// TIA Portal V16 export
// export: Created 2021-11-12T13:31:00.4796607Z, ExportSetting WithDefaults, DisplayName Totally Integrated Automation Portal, DisplayVersion V16 Update 3, DisplayName TIA Portal Version Control Interface, DisplayVersion V16 Update 2, DisplayName TIA Portal Openness, DisplayVersion V16 Update 3, DisplayName SINAMICS Startdrive Advanced, DisplayVersion V16 Update 5, DisplayName SINAMICS Startdrive G130, G150, S120, S150, SINAMICS MV, S210, DisplayVersion V16 Update 5, DisplayName SINAMICS Startdrive G110M, G120, G120C, G120D, G120P, G115D, DisplayVersion V16 Update 5, DisplayName STEP 7 Professional, DisplayVersion V16 Update 3, DisplayName STEP 7 Safety, DisplayVersion V16, DisplayName WinCC UA Professional, DisplayVersion V16 Update 3
FUNCTION_BLOCK "Safety_Aux"   // FB66, LAD
{ S7_Optimized_Access := 'TRUE' }
VERSION : 0.1
// stored: AutoNumber true, IsIECCheckEnabled false, IsRetainMemResEnabled false, MemoryReserve 100, SetENOAutomatically false, UDAEnableTagReadback false
   VAR
      "SF_100+RU01-QQ01" : "STD_EuchnerDoor";
      "SF_100+RU01-QQ02" { S7_SetPoint := 'True'} : "STD_EuchnerDoor";
      "SF_100+RU01-QQ03" { S7_SetPoint := 'True'} : "STD_EuchnerDoor";
      "SF_100+RU01-QQ04" { S7_SetPoint := 'True'} : "STD_EuchnerDoor";
      "SF_100+RU01-QQ05" { S7_SetPoint := 'True'} : "STD_EuchnerDoor";
      "SF_100+RU01-QQ06" { S7_SetPoint := 'True'} : "STD_EuchnerDoor";
      "SF_100+RU01-QQ07" { S7_SetPoint := 'True'} : "STD_EuchnerDoor";
      "SF_100+RU01-QQ08" { S7_SetPoint := 'True'} : "STD_EuchnerDoor";
      "SF_200+RU01-QQ01" { S7_SetPoint := 'True'} : "STD_EuchnerDoor";
      "SF_200+RU01-QQ02" { S7_SetPoint := 'True'} : "STD_EuchnerDoor";
      "SF_200+RU01-QQ03" { S7_SetPoint := 'True'} : "STD_EuchnerDoor";
      "SF_200+RU01-QQ04" { S7_SetPoint := 'True'} : "STD_EuchnerDoor";
      "SF_200+RU01-QQ05" { S7_SetPoint := 'True'} : "STD_EuchnerDoor";
      "SF_100+RU01-KF01" { S7_SetPoint := 'True'} : "STD_EuchnerSafetySwitch2MBM";
      "SF_100+RU01-KF02" { S7_SetPoint := 'True'} : "STD_EuchnerSafetySwitch2MBM";
      "SF_100+RU01-KF03" { S7_SetPoint := 'True'} : "STD_EuchnerSafetySwitch2MBM";
      "SF_200+RU01-KF01" { S7_SetPoint := 'True'} : "STD_EuchnerSafetySwitch2MBM";
      "SF_200+RU01-KF02" { S7_SetPoint := 'True'} : "STD_EuchnerSafetySwitch2MBM";
      "SF_200+RU01-KF03" { S7_SetPoint := 'True'} : "STD_EuchnerSafetySwitch2MBM";
      "SF_200+RU01-KF04" { S7_SetPoint := 'True'} : "STD_EuchnerSafetySwitch2MBM";
      SF_KAS1_ES { S7_SetPoint := 'True'} : "STD_DI_Mon";
      SF_KAS2_ES { S7_SetPoint := 'True'} : "STD_DI_Mon";
      SF_BSN1_2_ES { S7_SetPoint := 'True'} : "STD_DI_Mon";
      SF_BSN3_ES { S7_SetPoint := 'True'} : "STD_DI_Mon";
      SF_BSN4_5_ES { S7_SetPoint := 'True'} : "STD_DI_Mon";
      SF_SCH1_ES { S7_SetPoint := 'True'} : "STD_DI_Mon";
      SF_THM1_ES { S7_SetPoint := 'True'} : "STD_DI_Mon";
      SF_THM2_ES { S7_SetPoint := 'True'} : "STD_DI_Mon";
      "SF_000UH10-SF01_ES" { S7_SetPoint := 'True'} : "STD_DI_Mon";
      "SF_000UH11-SF01_ES" { S7_SetPoint := 'True'} : "STD_DI_Mon";
      "SF_100UH11-SF01_ES" { S7_SetPoint := 'True'} : "STD_DI_Mon";
      "SF_100UH12-SF01_ES" { S7_SetPoint := 'True'} : "STD_DI_Mon";
      "SF_100UH13-SF01_ES" { S7_SetPoint := 'True'} : "STD_DI_Mon";
      "SF_100UF01-SF01_ES" { S7_SetPoint := 'True'} : "STD_DI_Mon";
      "SF_200UH11-SF01_ES" { S7_SetPoint := 'True'} : "STD_DI_Mon";
      "SF_210UF01-SF01_ES" { S7_SetPoint := 'True'} : "STD_DI_Mon";
      "SF_220UF01-SF01_ES" { S7_SetPoint := 'True'} : "STD_DI_Mon";
      "SF_230UF01-SF01_ES" { S7_SetPoint := 'True'} : "STD_DI_Mon";
      "SF_200UF01-SF01_ES" { S7_SetPoint := 'True'} : "STD_DI_Mon";
      "SF_300UH11-SF01_ES" { S7_SetPoint := 'True'} : "STD_DI_Mon";
      "SF_310UH31-SF01_ES" { S7_SetPoint := 'True'} : "STD_DI_Mon";
      "SF_330UF01-SF01_ES" { S7_SetPoint := 'True'} : "STD_DI_Mon";
      "SF_400UH11-SF01_ES" { S7_SetPoint := 'True'} : "STD_DI_Mon";
      "SF_410UH31-SF01_ES" { S7_SetPoint := 'True'} : "STD_DI_Mon";
      "SF_420UH31-SF01_ES" { S7_SetPoint := 'True'} : "STD_DI_Mon";
      "SF_430UF01-SF01_ES" { S7_SetPoint := 'True'} : "STD_DI_Mon";
      SF_100QQ01_ES { S7_SetPoint := 'True'} : "STD_DI_Mon";
      SF_100QQ02_ES { S7_SetPoint := 'True'} : "STD_DI_Mon";
      SF_100QQ03_ES { S7_SetPoint := 'True'} : "STD_DI_Mon";
      SF_100QQ04_ES { S7_SetPoint := 'True'} : "STD_DI_Mon";
      SF_100QQ05_ES { S7_SetPoint := 'True'} : "STD_DI_Mon";
      SF_100QQ06_ES { S7_SetPoint := 'True'} : "STD_DI_Mon";
      SF_100QQ07_ES { S7_SetPoint := 'True'} : "STD_DI_Mon";
      SF_100QQ08_ES { S7_SetPoint := 'True'} : "STD_DI_Mon";
      SF_200QQ01_ES { S7_SetPoint := 'True'} : "STD_DI_Mon";
      SF_200QQ02_ES { S7_SetPoint := 'True'} : "STD_DI_Mon";
      SF_200QQ03_ES { S7_SetPoint := 'True'} : "STD_DI_Mon";
      SF_200QQ04_ES { S7_SetPoint := 'True'} : "STD_DI_Mon";
      SF_200QQ05_ES { S7_SetPoint := 'True'} : "STD_DI_Mon";
      SF_1R1RC01_ES { S7_SetPoint := 'True'} : "STD_DI_Mon";
      SF_1R2RC01_ES { S7_SetPoint := 'True'} : "STD_DI_Mon";
      SF_1R3RC01_ES { S7_SetPoint := 'True'} : "STD_DI_Mon";
      SF_1R4RC01_ES { S7_SetPoint := 'True'} : "STD_DI_Mon";
      SF_1R5RC01_ES { S7_SetPoint := 'True'} : "STD_DI_Mon";
      SF_1R6RC01_ES { S7_SetPoint := 'True'} : "STD_DI_Mon";
      SF_2R1RC01_ES { S7_SetPoint := 'True'} : "STD_DI_Mon";
      SF_2R2RC01_ES { S7_SetPoint := 'True'} : "STD_DI_Mon";
      "SF_000UH01-KF31" { S7_SetPoint := 'True'} : "STD_DI_Mon";
      "SF_000UH01-KF32" { S7_SetPoint := 'True'} : "STD_DI_Mon";
      "SF_000UH01-KF33" { S7_SetPoint := 'True'} : "STD_DI_Mon";
      "SF_000UH01-KF41" { S7_SetPoint := 'True'} : "STD_DI_Mon";
      "SF_000UH11-KF31" { S7_SetPoint := 'True'} : "STD_DI_Mon";
      "SF_000UH11-KF32" { S7_SetPoint := 'True'} : "STD_DI_Mon";
      "SF_100UH11-KF31" { S7_SetPoint := 'True'} : "STD_DI_Mon";
      "SF_100UH12-KF31" { S7_SetPoint := 'True'} : "STD_DI_Mon";
      "SF_100UH13-KF31" { S7_SetPoint := 'True'} : "STD_DI_Mon";
      "SF_100UH13-KF32" { S7_SetPoint := 'True'} : "STD_DI_Mon";
      "SF_200UH11-KF31" { S7_SetPoint := 'True'} : "STD_DI_Mon";
      "SF_300UH11-KF31" { S7_SetPoint := 'True'} : "STD_DI_Mon";
      "SF_310UH31-KF31" { S7_SetPoint := 'True'} : "STD_DI_Mon";
      "SF_400UH11-KF31" { S7_SetPoint := 'True'} : "STD_DI_Mon";
      "SF_410UH31-KF31" { S7_SetPoint := 'True'} : "STD_DI_Mon";
      "SF_420UH31-KF31" { S7_SetPoint := 'True'} : "STD_DI_Mon";
      "SF_100RU01-KF01" { S7_SetPoint := 'True'} : "STD_DI_Mon";
      "SF_100RU01-KF02" { S7_SetPoint := 'True'} : "STD_DI_Mon";
      "SF_100RU01-KF03" { S7_SetPoint := 'True'} : "STD_DI_Mon";
      "SF_200RU01-KF01" { S7_SetPoint := 'True'} : "STD_DI_Mon";
      "SF_200RU01-KF02" { S7_SetPoint := 'True'} : "STD_DI_Mon";
      "SF_200RU01-KF03" { S7_SetPoint := 'True'} : "STD_DI_Mon";
      "SF_200RU01-KF04" { S7_SetPoint := 'True'} : "STD_DI_Mon";
   END_VAR
   VAR_TEMP
      TS_AckSafety : "UDT_AckSafety1";   // Acknowledgement groups
      TB1UlckEn100 : Bool;
      TB1UlckEn101 : Bool;
      TB1UlckEn102 : Bool;
      TB1UlckEn103 : Bool;
      TB1UlckEn104 : Bool;
      TB1UlckEn105 : Bool;
      TB1UlckEn200 : Bool;
      TB1Fit1 : Bool;
   END_VAR
   VAR_TEMP   // added for the SCL form of the ladder/FBD networks
      _w1 : Bool;
      _w2 : Bool;
      _w3 : Bool;
      _w4 : Bool;
      _w5 : Bool;
      _w6 : Bool;
      _w7 : Bool;
      _w8 : Bool;
   END_VAR
BEGIN

REGION Network 1: *************** Resets ***************
END_REGION

REGION Network 2: Safety acknowledge Group01
   // Group01 - zone 100 buttons included panel 000-UH11, panel 000-UH10
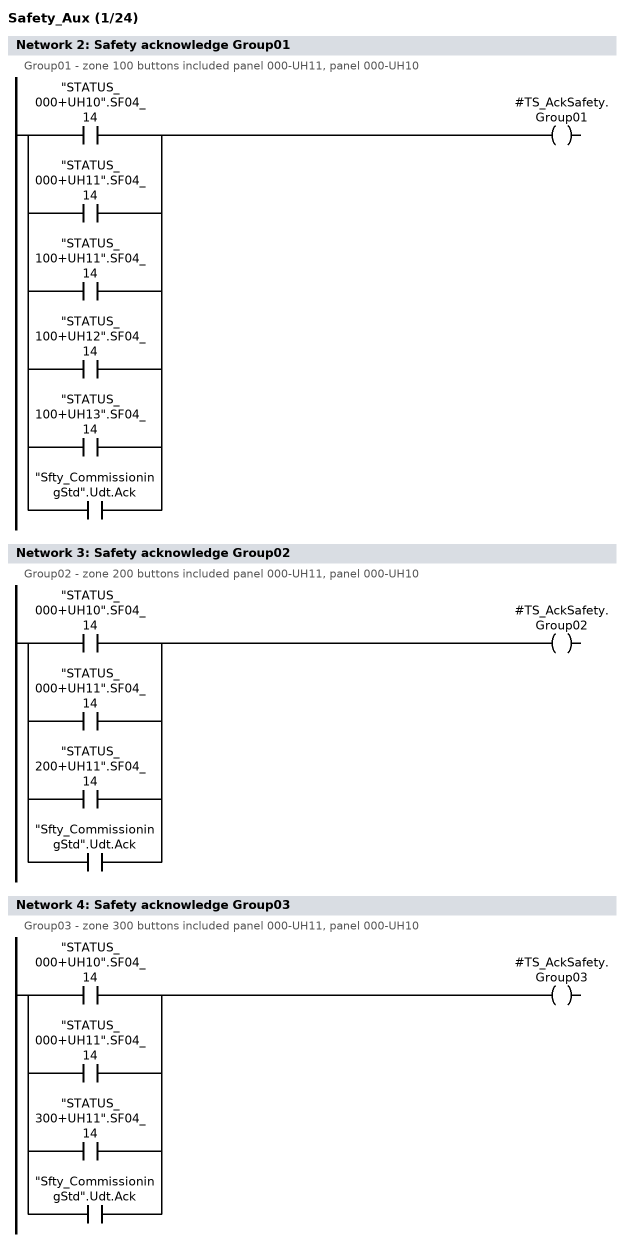
   RUNG wire#powerrail
      Contact( "STATUS_000+UH10".SF04_14 )
      wire#w1
      Coil( #TS_AckSafety.Group01 )
   END_RUNG
   RUNG wire#powerrail
      Contact( "STATUS_000+UH11".SF04_14 )
   END_RUNG wire#w1
   RUNG wire#powerrail
      Contact( "STATUS_100+UH11".SF04_14 )
   END_RUNG wire#w1
   RUNG wire#powerrail
      Contact( "STATUS_100+UH12".SF04_14 )
   END_RUNG wire#w1
   RUNG wire#powerrail
      Contact( "STATUS_100+UH13".SF04_14 )
   END_RUNG wire#w1
   RUNG wire#powerrail
      Contact( "Sfty_CommissioningStd".Udt.Ack )
   END_RUNG wire#w1
   // the same network as SCL:
   #TS_AckSafety.Group01 := "STATUS_000+UH10".SF04_14 OR "STATUS_000+UH11".SF04_14 OR "STATUS_100+UH11".SF04_14 OR "STATUS_100+UH12".SF04_14 OR "STATUS_100+UH13".SF04_14 OR "Sfty_CommissioningStd".Udt.Ack;
END_REGION

REGION Network 3: Safety acknowledge Group02
   // Group02 - zone 200 buttons included panel 000-UH11, panel 000-UH10
   RUNG wire#powerrail
      Contact( "STATUS_000+UH10".SF04_14 )
      wire#w1
      Coil( #TS_AckSafety.Group02 )
   END_RUNG
   RUNG wire#powerrail
      Contact( "STATUS_000+UH11".SF04_14 )
   END_RUNG wire#w1
   RUNG wire#powerrail
      Contact( "STATUS_200+UH11".SF04_14 )
   END_RUNG wire#w1
   RUNG wire#powerrail
      Contact( "Sfty_CommissioningStd".Udt.Ack )
   END_RUNG wire#w1
   // the same network as SCL:
   #TS_AckSafety.Group02 := "STATUS_000+UH10".SF04_14 OR "STATUS_000+UH11".SF04_14 OR "STATUS_200+UH11".SF04_14 OR "Sfty_CommissioningStd".Udt.Ack;
END_REGION

REGION Network 4: Safety acknowledge Group03
   // Group03 - zone 300 buttons included panel 000-UH11, panel 000-UH10
   RUNG wire#powerrail
      Contact( "STATUS_000+UH10".SF04_14 )
      wire#w1
      Coil( #TS_AckSafety.Group03 )
   END_RUNG
   RUNG wire#powerrail
      Contact( "STATUS_000+UH11".SF04_14 )
   END_RUNG wire#w1
   RUNG wire#powerrail
      Contact( "STATUS_300+UH11".SF04_14 )
   END_RUNG wire#w1
   RUNG wire#powerrail
      Contact( "Sfty_CommissioningStd".Udt.Ack )
   END_RUNG wire#w1
   // the same network as SCL:
   #TS_AckSafety.Group03 := "STATUS_000+UH10".SF04_14 OR "STATUS_000+UH11".SF04_14 OR "STATUS_300+UH11".SF04_14 OR "Sfty_CommissioningStd".Udt.Ack;
END_REGION

REGION Network 5: Safety acknowledge Group04
   // Group04 - zone 400 buttons included panel 000-UH11, panel 000-UH10
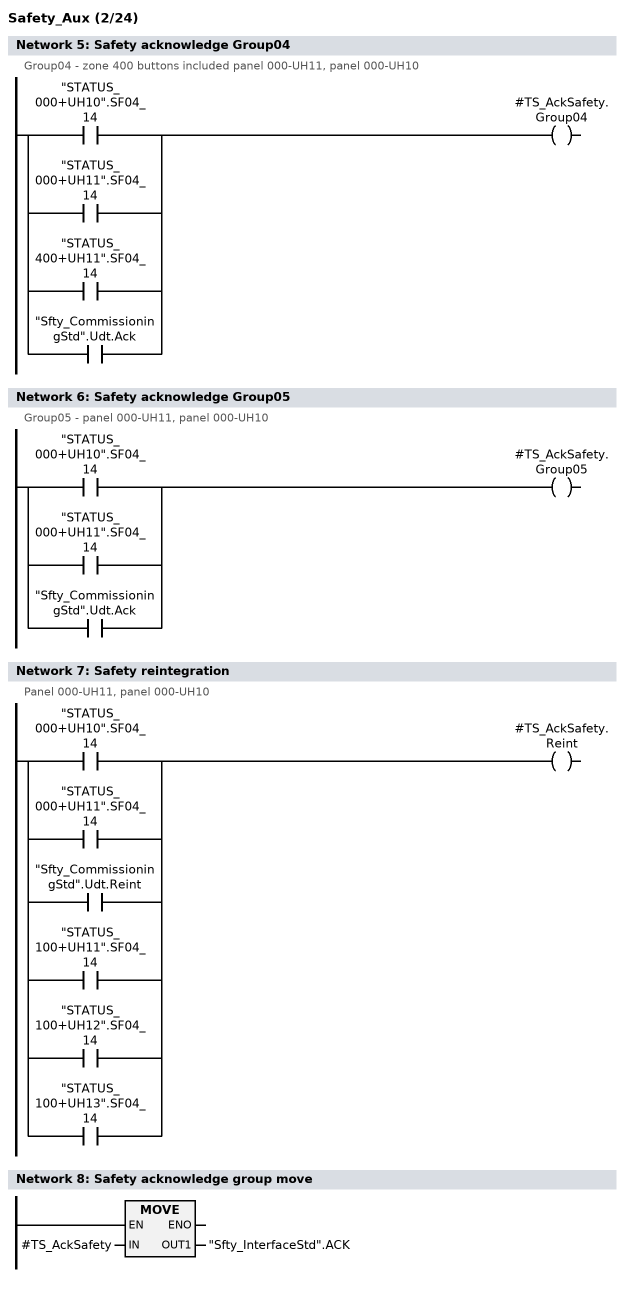
   RUNG wire#powerrail
      Contact( "STATUS_000+UH10".SF04_14 )
      wire#w1
      Coil( #TS_AckSafety.Group04 )
   END_RUNG
   RUNG wire#powerrail
      Contact( "STATUS_000+UH11".SF04_14 )
   END_RUNG wire#w1
   RUNG wire#powerrail
      Contact( "STATUS_400+UH11".SF04_14 )
   END_RUNG wire#w1
   RUNG wire#powerrail
      Contact( "Sfty_CommissioningStd".Udt.Ack )
   END_RUNG wire#w1
   // the same network as SCL:
   #TS_AckSafety.Group04 := "STATUS_000+UH10".SF04_14 OR "STATUS_000+UH11".SF04_14 OR "STATUS_400+UH11".SF04_14 OR "Sfty_CommissioningStd".Udt.Ack;
END_REGION

REGION Network 6: Safety acknowledge Group05
   // Group05 - panel 000-UH11, panel 000-UH10
   RUNG wire#powerrail
      Contact( "STATUS_000+UH10".SF04_14 )
      wire#w1
      Coil( #TS_AckSafety.Group05 )
   END_RUNG
   RUNG wire#powerrail
      Contact( "STATUS_000+UH11".SF04_14 )
   END_RUNG wire#w1
   RUNG wire#powerrail
      Contact( "Sfty_CommissioningStd".Udt.Ack )
   END_RUNG wire#w1
   // the same network as SCL:
   #TS_AckSafety.Group05 := "STATUS_000+UH10".SF04_14 OR "STATUS_000+UH11".SF04_14 OR "Sfty_CommissioningStd".Udt.Ack;
END_REGION

REGION Network 7: Safety reintegration
   // Panel 000-UH11, panel 000-UH10
   RUNG wire#powerrail
      Contact( "STATUS_000+UH10".SF04_14 )
      wire#w1
      Coil( #TS_AckSafety.Reint )
   END_RUNG
   RUNG wire#powerrail
      Contact( "STATUS_000+UH11".SF04_14 )
   END_RUNG wire#w1
   RUNG wire#powerrail
      Contact( "Sfty_CommissioningStd".Udt.Reint )
   END_RUNG wire#w1
   RUNG wire#powerrail
      Contact( "STATUS_100+UH11".SF04_14 )
   END_RUNG wire#w1
   RUNG wire#powerrail
      Contact( "STATUS_100+UH12".SF04_14 )
   END_RUNG wire#w1
   RUNG wire#powerrail
      Contact( "STATUS_100+UH13".SF04_14 )
   END_RUNG wire#w1
   // the same network as SCL:
   #TS_AckSafety.Reint := "STATUS_000+UH10".SF04_14 OR "STATUS_000+UH11".SF04_14 OR "Sfty_CommissioningStd".Udt.Reint OR "STATUS_100+UH11".SF04_14 OR "STATUS_100+UH12".SF04_14 OR "STATUS_100+UH13".SF04_14;
END_REGION

REGION Network 8: Safety acknowledge group move
   RUNG wire#powerrail
      Move(in := #TS_AckSafety, out1 => "Sfty_InterfaceStd".ACK)
   END_RUNG
   // the same network as SCL:
   "Sfty_InterfaceStd".ACK := #TS_AckSafety;
END_REGION

REGION Network 9: *************** Enable unlock gates ***************
END_REGION

REGION Network 10: Zone 100 - enable unlock gates
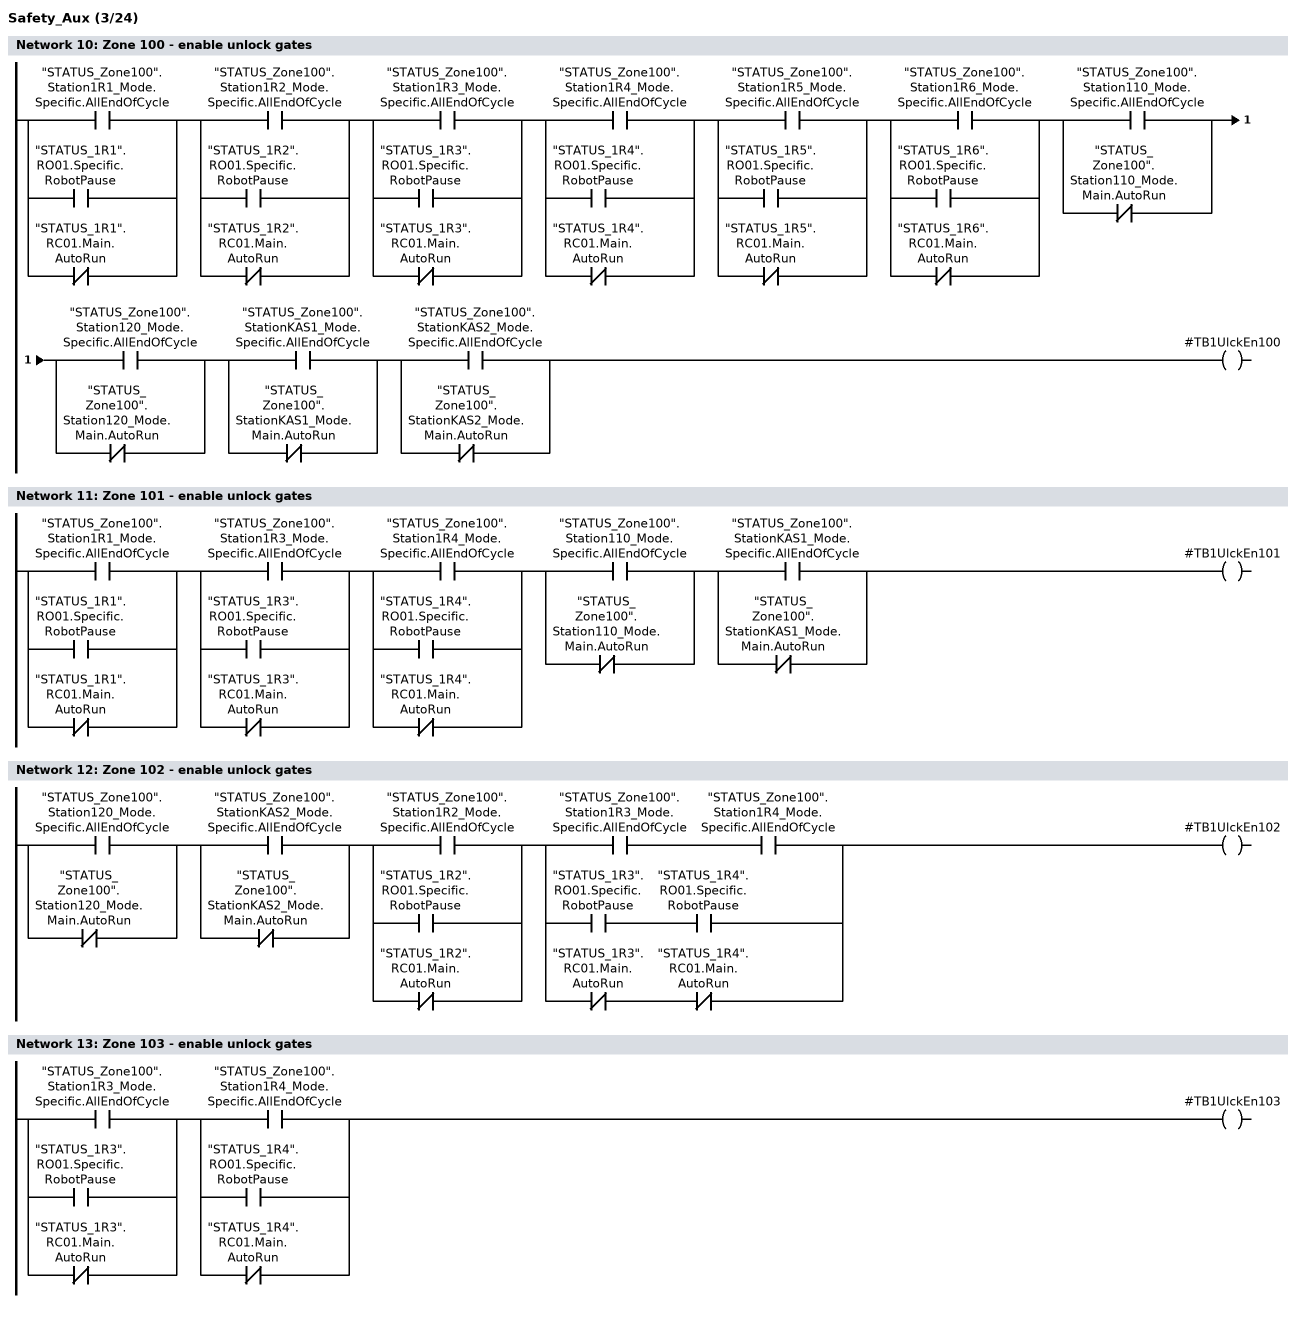
   RUNG wire#powerrail
      Contact( "STATUS_Zone100".Station1R1_Mode.Specific.AllEndOfCycle )
      wire#w1
      Contact( "STATUS_Zone100".Station1R2_Mode.Specific.AllEndOfCycle )
      wire#w2
      Contact( "STATUS_Zone100".Station1R3_Mode.Specific.AllEndOfCycle )
      wire#w3
      Contact( "STATUS_Zone100".Station1R4_Mode.Specific.AllEndOfCycle )
      wire#w4
      Contact( "STATUS_Zone100".Station1R5_Mode.Specific.AllEndOfCycle )
      wire#w5
      Contact( "STATUS_Zone100".Station1R6_Mode.Specific.AllEndOfCycle )
      wire#w6
      Contact( "STATUS_Zone100".Station110_Mode.Specific.AllEndOfCycle )
      wire#w7
      Contact( "STATUS_Zone100".Station120_Mode.Specific.AllEndOfCycle )
      wire#w8
      Contact( "STATUS_Zone100".StationKAS1_Mode.Specific.AllEndOfCycle )
      wire#w9
      Contact( "STATUS_Zone100".StationKAS2_Mode.Specific.AllEndOfCycle )
      wire#w10
      Coil( #TB1UlckEn100 )
   END_RUNG
   RUNG wire#powerrail
      Contact( "STATUS_1R1".RO01.Specific.RobotPause )
   END_RUNG wire#w1
   RUNG wire#powerrail
      I_Contact( "STATUS_1R1".RC01.Main.AutoRun )
   END_RUNG wire#w1
   RUNG wire#w1
      Contact( "STATUS_1R2".RO01.Specific.RobotPause )
   END_RUNG wire#w2
   RUNG wire#w1
      I_Contact( "STATUS_1R2".RC01.Main.AutoRun )
   END_RUNG wire#w2
   RUNG wire#w2
      Contact( "STATUS_1R3".RO01.Specific.RobotPause )
   END_RUNG wire#w3
   RUNG wire#w2
      I_Contact( "STATUS_1R3".RC01.Main.AutoRun )
   END_RUNG wire#w3
   RUNG wire#w3
      Contact( "STATUS_1R4".RO01.Specific.RobotPause )
   END_RUNG wire#w4
   RUNG wire#w3
      I_Contact( "STATUS_1R4".RC01.Main.AutoRun )
   END_RUNG wire#w4
   RUNG wire#w4
      Contact( "STATUS_1R5".RO01.Specific.RobotPause )
   END_RUNG wire#w5
   RUNG wire#w4
      I_Contact( "STATUS_1R5".RC01.Main.AutoRun )
   END_RUNG wire#w5
   RUNG wire#w5
      Contact( "STATUS_1R6".RO01.Specific.RobotPause )
   END_RUNG wire#w6
   RUNG wire#w5
      I_Contact( "STATUS_1R6".RC01.Main.AutoRun )
   END_RUNG wire#w6
   RUNG wire#w6
      I_Contact( "STATUS_Zone100".Station110_Mode.Main.AutoRun )
   END_RUNG wire#w7
   RUNG wire#w7
      I_Contact( "STATUS_Zone100".Station120_Mode.Main.AutoRun )
   END_RUNG wire#w8
   RUNG wire#w8
      I_Contact( "STATUS_Zone100".StationKAS1_Mode.Main.AutoRun )
   END_RUNG wire#w9
   RUNG wire#w9
      I_Contact( "STATUS_Zone100".StationKAS2_Mode.Main.AutoRun )
   END_RUNG wire#w10
   // the same network as SCL:
   #TB1UlckEn100 := ("STATUS_Zone100".Station1R1_Mode.Specific.AllEndOfCycle OR "STATUS_1R1".RO01.Specific.RobotPause OR NOT "STATUS_1R1".RC01.Main.AutoRun) AND ("STATUS_Zone100".Station1R2_Mode.Specific.AllEndOfCycle OR "STATUS_1R2".RO01.Specific.RobotPause OR NOT "STATUS_1R2".RC01.Main.AutoRun) AND ("STATUS_Zone100".Station1R3_Mode.Specific.AllEndOfCycle OR "STATUS_1R3".RO01.Specific.RobotPause OR NOT "STATUS_1R3".RC01.Main.AutoRun) AND ("STATUS_Zone100".Station1R4_Mode.Specific.AllEndOfCycle OR "STATUS_1R4".RO01.Specific.RobotPause OR NOT "STATUS_1R4".RC01.Main.AutoRun) AND ("STATUS_Zone100".Station1R5_Mode.Specific.AllEndOfCycle OR "STATUS_1R5".RO01.Specific.RobotPause OR NOT "STATUS_1R5".RC01.Main.AutoRun) AND ("STATUS_Zone100".Station1R6_Mode.Specific.AllEndOfCycle OR "STATUS_1R6".RO01.Specific.RobotPause OR NOT "STATUS_1R6".RC01.Main.AutoRun) AND ("STATUS_Zone100".Station110_Mode.Specific.AllEndOfCycle OR NOT "STATUS_Zone100".Station110_Mode.Main.AutoRun) AND ("STATUS_Zone100".Station120_Mode.Specific.AllEndOfCycle OR NOT "STATUS_Zone100".Station120_Mode.Main.AutoRun) AND ("STATUS_Zone100".StationKAS1_Mode.Specific.AllEndOfCycle OR NOT "STATUS_Zone100".StationKAS1_Mode.Main.AutoRun) AND ("STATUS_Zone100".StationKAS2_Mode.Specific.AllEndOfCycle OR NOT "STATUS_Zone100".StationKAS2_Mode.Main.AutoRun);
END_REGION

REGION Network 11: Zone 101 - enable unlock gates
   RUNG wire#powerrail
      Contact( "STATUS_Zone100".Station1R1_Mode.Specific.AllEndOfCycle )
      wire#w1
      Contact( "STATUS_Zone100".Station1R3_Mode.Specific.AllEndOfCycle )
      wire#w2
      Contact( "STATUS_Zone100".Station1R4_Mode.Specific.AllEndOfCycle )
      wire#w3
      Contact( "STATUS_Zone100".Station110_Mode.Specific.AllEndOfCycle )
      wire#w4
      Contact( "STATUS_Zone100".StationKAS1_Mode.Specific.AllEndOfCycle )
      wire#w5
      Coil( #TB1UlckEn101 )
   END_RUNG
   RUNG wire#powerrail
      Contact( "STATUS_1R1".RO01.Specific.RobotPause )
   END_RUNG wire#w1
   RUNG wire#powerrail
      I_Contact( "STATUS_1R1".RC01.Main.AutoRun )
   END_RUNG wire#w1
   RUNG wire#w1
      Contact( "STATUS_1R3".RO01.Specific.RobotPause )
   END_RUNG wire#w2
   RUNG wire#w1
      I_Contact( "STATUS_1R3".RC01.Main.AutoRun )
   END_RUNG wire#w2
   RUNG wire#w2
      Contact( "STATUS_1R4".RO01.Specific.RobotPause )
   END_RUNG wire#w3
   RUNG wire#w2
      I_Contact( "STATUS_1R4".RC01.Main.AutoRun )
   END_RUNG wire#w3
   RUNG wire#w3
      I_Contact( "STATUS_Zone100".Station110_Mode.Main.AutoRun )
   END_RUNG wire#w4
   RUNG wire#w4
      I_Contact( "STATUS_Zone100".StationKAS1_Mode.Main.AutoRun )
   END_RUNG wire#w5
   // the same network as SCL:
   #TB1UlckEn101 := ("STATUS_Zone100".Station1R1_Mode.Specific.AllEndOfCycle OR "STATUS_1R1".RO01.Specific.RobotPause OR NOT "STATUS_1R1".RC01.Main.AutoRun) AND ("STATUS_Zone100".Station1R3_Mode.Specific.AllEndOfCycle OR "STATUS_1R3".RO01.Specific.RobotPause OR NOT "STATUS_1R3".RC01.Main.AutoRun) AND ("STATUS_Zone100".Station1R4_Mode.Specific.AllEndOfCycle OR "STATUS_1R4".RO01.Specific.RobotPause OR NOT "STATUS_1R4".RC01.Main.AutoRun) AND ("STATUS_Zone100".Station110_Mode.Specific.AllEndOfCycle OR NOT "STATUS_Zone100".Station110_Mode.Main.AutoRun) AND ("STATUS_Zone100".StationKAS1_Mode.Specific.AllEndOfCycle OR NOT "STATUS_Zone100".StationKAS1_Mode.Main.AutoRun);
END_REGION

REGION Network 12: Zone 102 - enable unlock gates
   RUNG wire#powerrail
      Contact( "STATUS_Zone100".Station120_Mode.Specific.AllEndOfCycle )
      wire#w1
      Contact( "STATUS_Zone100".StationKAS2_Mode.Specific.AllEndOfCycle )
      wire#w2
      Contact( "STATUS_Zone100".Station1R2_Mode.Specific.AllEndOfCycle )
      wire#w3
      Contact( "STATUS_Zone100".Station1R3_Mode.Specific.AllEndOfCycle )
      Contact( "STATUS_Zone100".Station1R4_Mode.Specific.AllEndOfCycle )
      wire#w4
      Coil( #TB1UlckEn102 )
   END_RUNG
   RUNG wire#powerrail
      I_Contact( "STATUS_Zone100".Station120_Mode.Main.AutoRun )
   END_RUNG wire#w1
   RUNG wire#w1
      I_Contact( "STATUS_Zone100".StationKAS2_Mode.Main.AutoRun )
   END_RUNG wire#w2
   RUNG wire#w2
      Contact( "STATUS_1R2".RO01.Specific.RobotPause )
   END_RUNG wire#w3
   RUNG wire#w2
      I_Contact( "STATUS_1R2".RC01.Main.AutoRun )
   END_RUNG wire#w3
   RUNG wire#w3
      Contact( "STATUS_1R3".RO01.Specific.RobotPause )
      Contact( "STATUS_1R4".RO01.Specific.RobotPause )
   END_RUNG wire#w4
   RUNG wire#w3
      I_Contact( "STATUS_1R3".RC01.Main.AutoRun )
      I_Contact( "STATUS_1R4".RC01.Main.AutoRun )
   END_RUNG wire#w4
   // the same network as SCL:
   #TB1UlckEn102 := ("STATUS_Zone100".Station120_Mode.Specific.AllEndOfCycle OR NOT "STATUS_Zone100".Station120_Mode.Main.AutoRun) AND ("STATUS_Zone100".StationKAS2_Mode.Specific.AllEndOfCycle OR NOT "STATUS_Zone100".StationKAS2_Mode.Main.AutoRun) AND ("STATUS_Zone100".Station1R2_Mode.Specific.AllEndOfCycle OR "STATUS_1R2".RO01.Specific.RobotPause OR NOT "STATUS_1R2".RC01.Main.AutoRun) AND (("STATUS_Zone100".Station1R3_Mode.Specific.AllEndOfCycle AND "STATUS_Zone100".Station1R4_Mode.Specific.AllEndOfCycle) OR ("STATUS_1R3".RO01.Specific.RobotPause AND "STATUS_1R4".RO01.Specific.RobotPause) OR (NOT "STATUS_1R3".RC01.Main.AutoRun AND NOT "STATUS_1R4".RC01.Main.AutoRun));
END_REGION

REGION Network 13: Zone 103 - enable unlock gates
   RUNG wire#powerrail
      Contact( "STATUS_Zone100".Station1R3_Mode.Specific.AllEndOfCycle )
      wire#w1
      Contact( "STATUS_Zone100".Station1R4_Mode.Specific.AllEndOfCycle )
      wire#w2
      Coil( #TB1UlckEn103 )
   END_RUNG
   RUNG wire#powerrail
      Contact( "STATUS_1R3".RO01.Specific.RobotPause )
   END_RUNG wire#w1
   RUNG wire#powerrail
      I_Contact( "STATUS_1R3".RC01.Main.AutoRun )
   END_RUNG wire#w1
   RUNG wire#w1
      Contact( "STATUS_1R4".RO01.Specific.RobotPause )
   END_RUNG wire#w2
   RUNG wire#w1
      I_Contact( "STATUS_1R4".RC01.Main.AutoRun )
   END_RUNG wire#w2
   // the same network as SCL:
   #TB1UlckEn103 := ("STATUS_Zone100".Station1R3_Mode.Specific.AllEndOfCycle OR "STATUS_1R3".RO01.Specific.RobotPause OR NOT "STATUS_1R3".RC01.Main.AutoRun) AND ("STATUS_Zone100".Station1R4_Mode.Specific.AllEndOfCycle OR "STATUS_1R4".RO01.Specific.RobotPause OR NOT "STATUS_1R4".RC01.Main.AutoRun);
END_REGION

REGION Network 14: Zone 104 - enable unlock gates
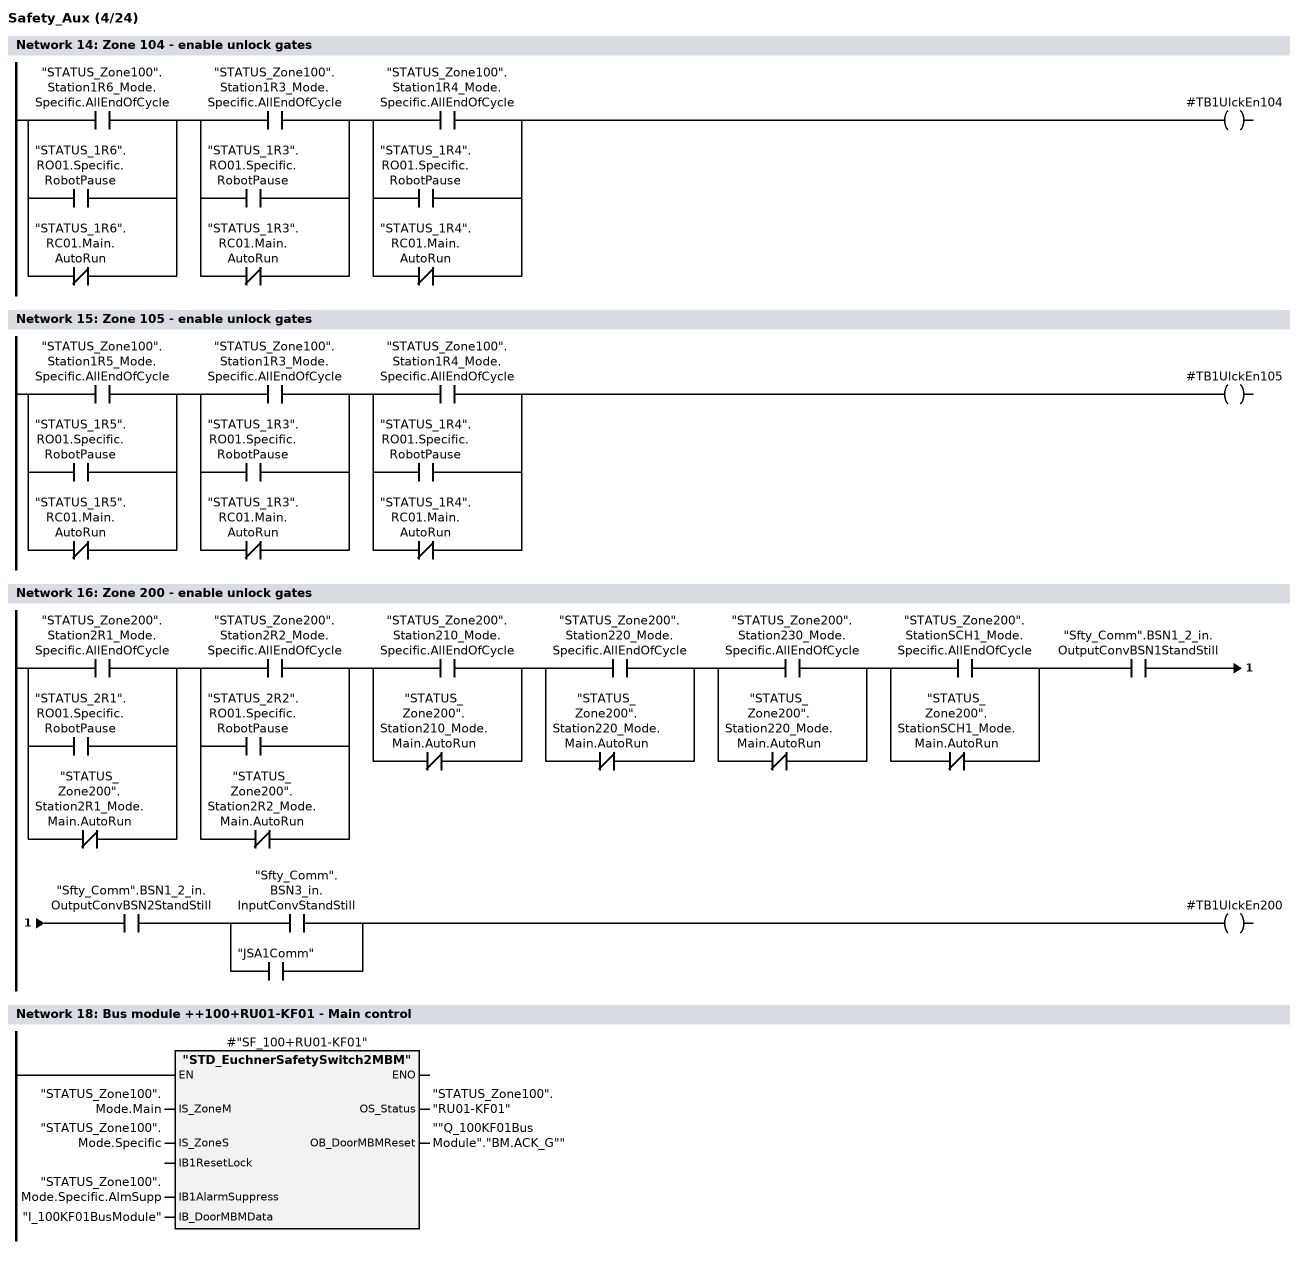
   RUNG wire#powerrail
      Contact( "STATUS_Zone100".Station1R6_Mode.Specific.AllEndOfCycle )
      wire#w1
      Contact( "STATUS_Zone100".Station1R3_Mode.Specific.AllEndOfCycle )
      wire#w2
      Contact( "STATUS_Zone100".Station1R4_Mode.Specific.AllEndOfCycle )
      wire#w3
      Coil( #TB1UlckEn104 )
   END_RUNG
   RUNG wire#powerrail
      Contact( "STATUS_1R6".RO01.Specific.RobotPause )
   END_RUNG wire#w1
   RUNG wire#powerrail
      I_Contact( "STATUS_1R6".RC01.Main.AutoRun )
   END_RUNG wire#w1
   RUNG wire#w1
      Contact( "STATUS_1R3".RO01.Specific.RobotPause )
   END_RUNG wire#w2
   RUNG wire#w1
      I_Contact( "STATUS_1R3".RC01.Main.AutoRun )
   END_RUNG wire#w2
   RUNG wire#w2
      Contact( "STATUS_1R4".RO01.Specific.RobotPause )
   END_RUNG wire#w3
   RUNG wire#w2
      I_Contact( "STATUS_1R4".RC01.Main.AutoRun )
   END_RUNG wire#w3
   // the same network as SCL:
   #TB1UlckEn104 := ("STATUS_Zone100".Station1R6_Mode.Specific.AllEndOfCycle OR "STATUS_1R6".RO01.Specific.RobotPause OR NOT "STATUS_1R6".RC01.Main.AutoRun) AND ("STATUS_Zone100".Station1R3_Mode.Specific.AllEndOfCycle OR "STATUS_1R3".RO01.Specific.RobotPause OR NOT "STATUS_1R3".RC01.Main.AutoRun) AND ("STATUS_Zone100".Station1R4_Mode.Specific.AllEndOfCycle OR "STATUS_1R4".RO01.Specific.RobotPause OR NOT "STATUS_1R4".RC01.Main.AutoRun);
END_REGION

REGION Network 15: Zone 105 - enable unlock gates
   RUNG wire#powerrail
      Contact( "STATUS_Zone100".Station1R5_Mode.Specific.AllEndOfCycle )
      wire#w1
      Contact( "STATUS_Zone100".Station1R3_Mode.Specific.AllEndOfCycle )
      wire#w2
      Contact( "STATUS_Zone100".Station1R4_Mode.Specific.AllEndOfCycle )
      wire#w3
      Coil( #TB1UlckEn105 )
   END_RUNG
   RUNG wire#powerrail
      Contact( "STATUS_1R5".RO01.Specific.RobotPause )
   END_RUNG wire#w1
   RUNG wire#powerrail
      I_Contact( "STATUS_1R5".RC01.Main.AutoRun )
   END_RUNG wire#w1
   RUNG wire#w1
      Contact( "STATUS_1R3".RO01.Specific.RobotPause )
   END_RUNG wire#w2
   RUNG wire#w1
      I_Contact( "STATUS_1R3".RC01.Main.AutoRun )
   END_RUNG wire#w2
   RUNG wire#w2
      Contact( "STATUS_1R4".RO01.Specific.RobotPause )
   END_RUNG wire#w3
   RUNG wire#w2
      I_Contact( "STATUS_1R4".RC01.Main.AutoRun )
   END_RUNG wire#w3
   // the same network as SCL:
   #TB1UlckEn105 := ("STATUS_Zone100".Station1R5_Mode.Specific.AllEndOfCycle OR "STATUS_1R5".RO01.Specific.RobotPause OR NOT "STATUS_1R5".RC01.Main.AutoRun) AND ("STATUS_Zone100".Station1R3_Mode.Specific.AllEndOfCycle OR "STATUS_1R3".RO01.Specific.RobotPause OR NOT "STATUS_1R3".RC01.Main.AutoRun) AND ("STATUS_Zone100".Station1R4_Mode.Specific.AllEndOfCycle OR "STATUS_1R4".RO01.Specific.RobotPause OR NOT "STATUS_1R4".RC01.Main.AutoRun);
END_REGION

REGION Network 16: Zone 200 - enable unlock gates
   RUNG wire#powerrail
      Contact( "STATUS_Zone200".Station2R1_Mode.Specific.AllEndOfCycle )
      wire#w1
      Contact( "STATUS_Zone200".Station2R2_Mode.Specific.AllEndOfCycle )
      wire#w2
      Contact( "STATUS_Zone200".Station210_Mode.Specific.AllEndOfCycle )
      wire#w3
      Contact( "STATUS_Zone200".Station220_Mode.Specific.AllEndOfCycle )
      wire#w4
      Contact( "STATUS_Zone200".Station230_Mode.Specific.AllEndOfCycle )
      wire#w5
      Contact( "STATUS_Zone200".StationSCH1_Mode.Specific.AllEndOfCycle )
      wire#w6
      Contact( "Sfty_Comm".BSN1_2_in.OutputConvBSN1StandStill )
      Contact( "Sfty_Comm".BSN1_2_in.OutputConvBSN2StandStill )
      wire#w7
      Contact( "Sfty_Comm".BSN3_in.InputConvStandStill )
      wire#w8
      Coil( #TB1UlckEn200 )
   END_RUNG
   RUNG wire#powerrail
      Contact( "STATUS_2R1".RO01.Specific.RobotPause )
   END_RUNG wire#w1
   RUNG wire#powerrail
      I_Contact( "STATUS_Zone200".Station2R1_Mode.Main.AutoRun )
   END_RUNG wire#w1
   RUNG wire#w1
      Contact( "STATUS_2R2".RO01.Specific.RobotPause )
   END_RUNG wire#w2
   RUNG wire#w1
      I_Contact( "STATUS_Zone200".Station2R2_Mode.Main.AutoRun )
   END_RUNG wire#w2
   RUNG wire#w2
      I_Contact( "STATUS_Zone200".Station210_Mode.Main.AutoRun )
   END_RUNG wire#w3
   RUNG wire#w3
      I_Contact( "STATUS_Zone200".Station220_Mode.Main.AutoRun )
   END_RUNG wire#w4
   RUNG wire#w4
      I_Contact( "STATUS_Zone200".Station220_Mode.Main.AutoRun )
   END_RUNG wire#w5
   RUNG wire#w5
      I_Contact( "STATUS_Zone200".StationSCH1_Mode.Main.AutoRun )
   END_RUNG wire#w6
   RUNG wire#w7
      Contact( "JSA1Comm" )
   END_RUNG wire#w8
   // the same network as SCL:
   #TB1UlckEn200 := ("STATUS_Zone200".Station2R1_Mode.Specific.AllEndOfCycle OR "STATUS_2R1".RO01.Specific.RobotPause OR NOT "STATUS_Zone200".Station2R1_Mode.Main.AutoRun) AND ("STATUS_Zone200".Station2R2_Mode.Specific.AllEndOfCycle OR "STATUS_2R2".RO01.Specific.RobotPause OR NOT "STATUS_Zone200".Station2R2_Mode.Main.AutoRun) AND ("STATUS_Zone200".Station210_Mode.Specific.AllEndOfCycle OR NOT "STATUS_Zone200".Station210_Mode.Main.AutoRun) AND ("STATUS_Zone200".Station220_Mode.Specific.AllEndOfCycle OR NOT "STATUS_Zone200".Station220_Mode.Main.AutoRun) AND ("STATUS_Zone200".Station230_Mode.Specific.AllEndOfCycle OR NOT "STATUS_Zone200".Station220_Mode.Main.AutoRun) AND ("STATUS_Zone200".StationSCH1_Mode.Specific.AllEndOfCycle OR NOT "STATUS_Zone200".StationSCH1_Mode.Main.AutoRun) AND "Sfty_Comm".BSN1_2_in.OutputConvBSN1StandStill AND "Sfty_Comm".BSN1_2_in.OutputConvBSN2StandStill AND ("Sfty_Comm".BSN3_in.InputConvStandStill OR "JSA1Comm");
END_REGION

REGION Network 17: *************** Gate controls ***************
END_REGION

REGION Network 18: Bus module ++100+RU01-KF01 - Main control
   RUNG wire#powerrail
      #"SF_100+RU01-KF01"(IS_ZoneM := "STATUS_Zone100".Mode.Main, IS_ZoneS := "STATUS_Zone100".Mode.Specific, IB1ResetLock :=, IB1AlarmSuppress := "STATUS_Zone100".Mode.Specific.AlmSupp, IB_DoorMBMData := "I_100KF01BusModule", OS_Status => "STATUS_Zone100"."RU01-KF01", OB_DoorMBMReset => ""Q_100KF01BusModule"."BM.ACK_G"")
   END_RUNG
   // the same network as SCL:
   // no checked SCL form for this network; see the picture
END_REGION

REGION Network 19: Bus module ++100+RU01-KF02 - Main control
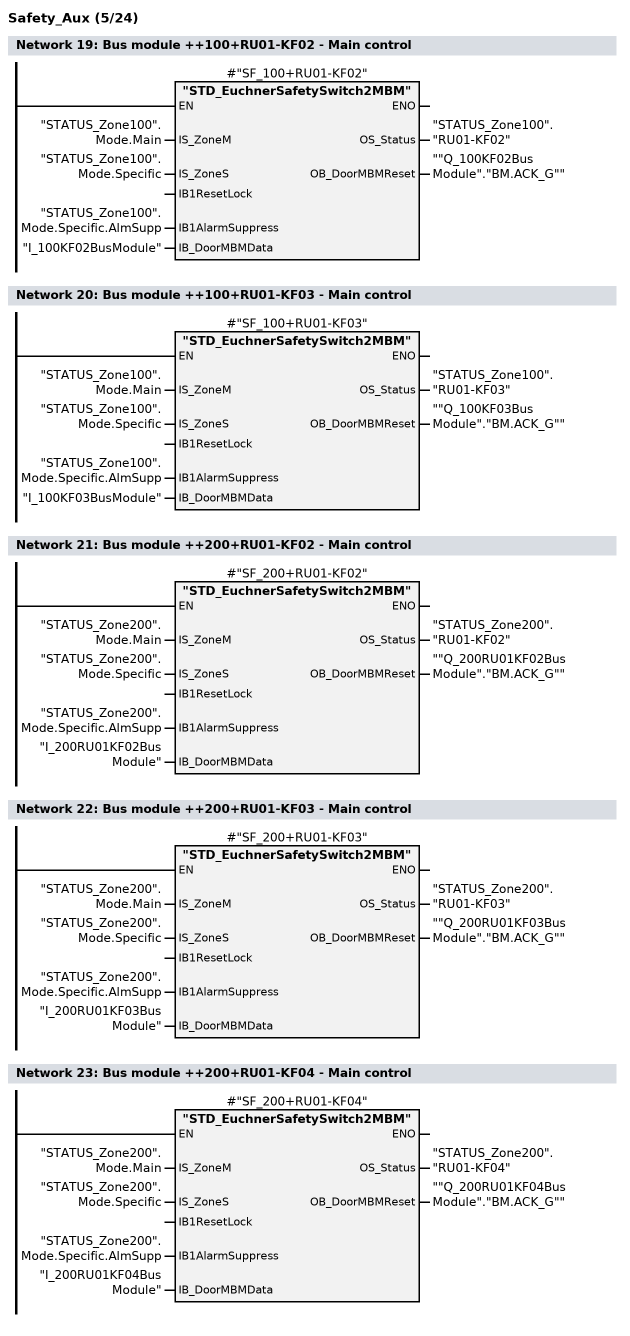
   RUNG wire#powerrail
      #"SF_100+RU01-KF02"(IS_ZoneM := "STATUS_Zone100".Mode.Main, IS_ZoneS := "STATUS_Zone100".Mode.Specific, IB1ResetLock :=, IB1AlarmSuppress := "STATUS_Zone100".Mode.Specific.AlmSupp, IB_DoorMBMData := "I_100KF02BusModule", OS_Status => "STATUS_Zone100"."RU01-KF02", OB_DoorMBMReset => ""Q_100KF02BusModule"."BM.ACK_G"")
   END_RUNG
   // the same network as SCL:
   // no checked SCL form for this network; see the picture
END_REGION

REGION Network 20: Bus module ++100+RU01-KF03 - Main control
   RUNG wire#powerrail
      #"SF_100+RU01-KF03"(IS_ZoneM := "STATUS_Zone100".Mode.Main, IS_ZoneS := "STATUS_Zone100".Mode.Specific, IB1ResetLock :=, IB1AlarmSuppress := "STATUS_Zone100".Mode.Specific.AlmSupp, IB_DoorMBMData := "I_100KF03BusModule", OS_Status => "STATUS_Zone100"."RU01-KF03", OB_DoorMBMReset => ""Q_100KF03BusModule"."BM.ACK_G"")
   END_RUNG
   // the same network as SCL:
   // no checked SCL form for this network; see the picture
END_REGION

REGION Network 21: Bus module ++200+RU01-KF02 - Main control
   RUNG wire#powerrail
      #"SF_200+RU01-KF02"(IS_ZoneM := "STATUS_Zone200".Mode.Main, IS_ZoneS := "STATUS_Zone200".Mode.Specific, IB1ResetLock :=, IB1AlarmSuppress := "STATUS_Zone200".Mode.Specific.AlmSupp, IB_DoorMBMData := "I_200RU01KF02BusModule", OS_Status => "STATUS_Zone200"."RU01-KF02", OB_DoorMBMReset => ""Q_200RU01KF02BusModule"."BM.ACK_G"")
   END_RUNG
   // the same network as SCL:
   // no checked SCL form for this network; see the picture
END_REGION

REGION Network 22: Bus module ++200+RU01-KF03 - Main control
   RUNG wire#powerrail
      #"SF_200+RU01-KF03"(IS_ZoneM := "STATUS_Zone200".Mode.Main, IS_ZoneS := "STATUS_Zone200".Mode.Specific, IB1ResetLock :=, IB1AlarmSuppress := "STATUS_Zone200".Mode.Specific.AlmSupp, IB_DoorMBMData := "I_200RU01KF03BusModule", OS_Status => "STATUS_Zone200"."RU01-KF03", OB_DoorMBMReset => ""Q_200RU01KF03BusModule"."BM.ACK_G"")
   END_RUNG
   // the same network as SCL:
   // no checked SCL form for this network; see the picture
END_REGION

REGION Network 23: Bus module ++200+RU01-KF04 - Main control
   RUNG wire#powerrail
      #"SF_200+RU01-KF04"(IS_ZoneM := "STATUS_Zone200".Mode.Main, IS_ZoneS := "STATUS_Zone200".Mode.Specific, IB1ResetLock :=, IB1AlarmSuppress := "STATUS_Zone200".Mode.Specific.AlmSupp, IB_DoorMBMData := "I_200RU01KF04BusModule", OS_Status => "STATUS_Zone200"."RU01-KF04", OB_DoorMBMReset => ""Q_200RU01KF04BusModule"."BM.ACK_G"")
   END_RUNG
   // the same network as SCL:
   // no checked SCL form for this network; see the picture
END_REGION

REGION Network 24: Lock module ++100+RU01-QQ01 - Main control
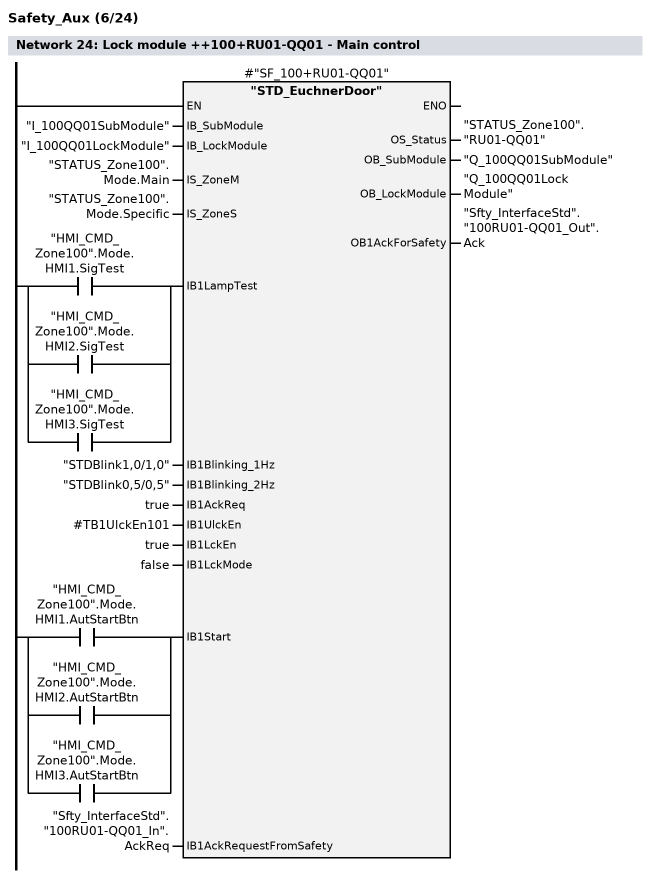
   RUNG wire#powerrail
      #"SF_100+RU01-QQ01"(IB1LampTest := wire#w1, IB1Start := wire#w2, IB_SubModule := "I_100QQ01SubModule", IB_LockModule := "I_100QQ01LockModule", IS_ZoneM := "STATUS_Zone100".Mode.Main, IS_ZoneS := "STATUS_Zone100".Mode.Specific, IB1Blinking_1Hz := "STDBlink1,0/1,0", IB1Blinking_2Hz := "STDBlink0,5/0,5", IB1AckReq := true, IB1UlckEn := #TB1UlckEn101, IB1LckEn := true, IB1LckMode := false, IB1AckRequestFromSafety := "Sfty_InterfaceStd"."100RU01-QQ01_In".AckReq, OS_Status => "STATUS_Zone100"."RU01-QQ01", OB_SubModule => "Q_100QQ01SubModule", OB_LockModule => "Q_100QQ01LockModule", OB1AckForSafety => "Sfty_InterfaceStd"."100RU01-QQ01_Out".Ack)
   END_RUNG
   RUNG wire#powerrail
      Contact( "HMI_CMD_Zone100".Mode.HMI1.SigTest )
   END_RUNG wire#w1
   RUNG wire#powerrail
      Contact( "HMI_CMD_Zone100".Mode.HMI2.SigTest )
   END_RUNG wire#w1
   RUNG wire#powerrail
      Contact( "HMI_CMD_Zone100".Mode.HMI3.SigTest )
   END_RUNG wire#w1
   RUNG wire#powerrail
      Contact( "HMI_CMD_Zone100".Mode.HMI1.AutStartBtn )
   END_RUNG wire#w2
   RUNG wire#powerrail
      Contact( "HMI_CMD_Zone100".Mode.HMI2.AutStartBtn )
   END_RUNG wire#w2
   RUNG wire#powerrail
      Contact( "HMI_CMD_Zone100".Mode.HMI3.AutStartBtn )
   END_RUNG wire#w2
   // the same network as SCL:
   #"SF_100+RU01-QQ01"(IB_SubModule := "I_100QQ01SubModule",   // "STD_EuchnerDoor"
                       IB_LockModule := "I_100QQ01LockModule",
                       IS_ZoneM := "STATUS_Zone100".Mode.Main,
                       IS_ZoneS := "STATUS_Zone100".Mode.Specific,
                       IB1LampTest := "HMI_CMD_Zone100".Mode.HMI1.SigTest OR "HMI_CMD_Zone100".Mode.HMI2.SigTest OR "HMI_CMD_Zone100".Mode.HMI3.SigTest,
                       IB1Blinking_1Hz := "STDBlink1,0/1,0",
                       IB1Blinking_2Hz := "STDBlink0,5/0,5",
                       IB1AckReq := true,
                       IB1UlckEn := #TB1UlckEn101,
                       IB1LckEn := true,
                       IB1LckMode := false,
                       IB1Start := "HMI_CMD_Zone100".Mode.HMI1.AutStartBtn OR "HMI_CMD_Zone100".Mode.HMI2.AutStartBtn OR "HMI_CMD_Zone100".Mode.HMI3.AutStartBtn,
                       IB1AckRequestFromSafety := "Sfty_InterfaceStd"."100RU01-QQ01_In".AckReq,
                       OS_Status => "STATUS_Zone100"."RU01-QQ01",
                       OB_SubModule => "Q_100QQ01SubModule",
                       OB_LockModule => "Q_100QQ01LockModule",
                       OB1AckForSafety => "Sfty_InterfaceStd"."100RU01-QQ01_Out".Ack);
END_REGION

REGION Network 25: Lock module ++100+RU01-QQ02 - Main control
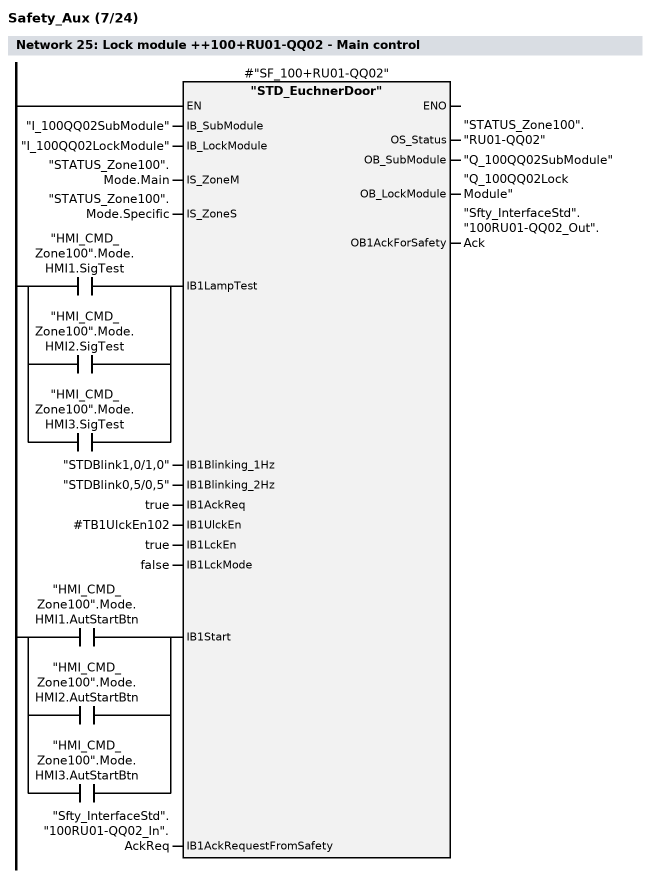
   RUNG wire#powerrail
      #"SF_100+RU01-QQ02"(IB1LampTest := wire#w1, IB1Start := wire#w2, IB_SubModule := "I_100QQ02SubModule", IB_LockModule := "I_100QQ02LockModule", IS_ZoneM := "STATUS_Zone100".Mode.Main, IS_ZoneS := "STATUS_Zone100".Mode.Specific, IB1Blinking_1Hz := "STDBlink1,0/1,0", IB1Blinking_2Hz := "STDBlink0,5/0,5", IB1AckReq := true, IB1UlckEn := #TB1UlckEn102, IB1LckEn := true, IB1LckMode := false, IB1AckRequestFromSafety := "Sfty_InterfaceStd"."100RU01-QQ02_In".AckReq, OS_Status => "STATUS_Zone100"."RU01-QQ02", OB_SubModule => "Q_100QQ02SubModule", OB_LockModule => "Q_100QQ02LockModule", OB1AckForSafety => "Sfty_InterfaceStd"."100RU01-QQ02_Out".Ack)
   END_RUNG
   RUNG wire#powerrail
      Contact( "HMI_CMD_Zone100".Mode.HMI1.SigTest )
   END_RUNG wire#w1
   RUNG wire#powerrail
      Contact( "HMI_CMD_Zone100".Mode.HMI2.SigTest )
   END_RUNG wire#w1
   RUNG wire#powerrail
      Contact( "HMI_CMD_Zone100".Mode.HMI3.SigTest )
   END_RUNG wire#w1
   RUNG wire#powerrail
      Contact( "HMI_CMD_Zone100".Mode.HMI1.AutStartBtn )
   END_RUNG wire#w2
   RUNG wire#powerrail
      Contact( "HMI_CMD_Zone100".Mode.HMI2.AutStartBtn )
   END_RUNG wire#w2
   RUNG wire#powerrail
      Contact( "HMI_CMD_Zone100".Mode.HMI3.AutStartBtn )
   END_RUNG wire#w2
   // the same network as SCL:
   #"SF_100+RU01-QQ02"(IB_SubModule := "I_100QQ02SubModule",   // "STD_EuchnerDoor"
                       IB_LockModule := "I_100QQ02LockModule",
                       IS_ZoneM := "STATUS_Zone100".Mode.Main,
                       IS_ZoneS := "STATUS_Zone100".Mode.Specific,
                       IB1LampTest := "HMI_CMD_Zone100".Mode.HMI1.SigTest OR "HMI_CMD_Zone100".Mode.HMI2.SigTest OR "HMI_CMD_Zone100".Mode.HMI3.SigTest,
                       IB1Blinking_1Hz := "STDBlink1,0/1,0",
                       IB1Blinking_2Hz := "STDBlink0,5/0,5",
                       IB1AckReq := true,
                       IB1UlckEn := #TB1UlckEn102,
                       IB1LckEn := true,
                       IB1LckMode := false,
                       IB1Start := "HMI_CMD_Zone100".Mode.HMI1.AutStartBtn OR "HMI_CMD_Zone100".Mode.HMI2.AutStartBtn OR "HMI_CMD_Zone100".Mode.HMI3.AutStartBtn,
                       IB1AckRequestFromSafety := "Sfty_InterfaceStd"."100RU01-QQ02_In".AckReq,
                       OS_Status => "STATUS_Zone100"."RU01-QQ02",
                       OB_SubModule => "Q_100QQ02SubModule",
                       OB_LockModule => "Q_100QQ02LockModule",
                       OB1AckForSafety => "Sfty_InterfaceStd"."100RU01-QQ02_Out".Ack);
END_REGION

REGION Network 26: Lock module ++100+RU01-QQ03 - Main control
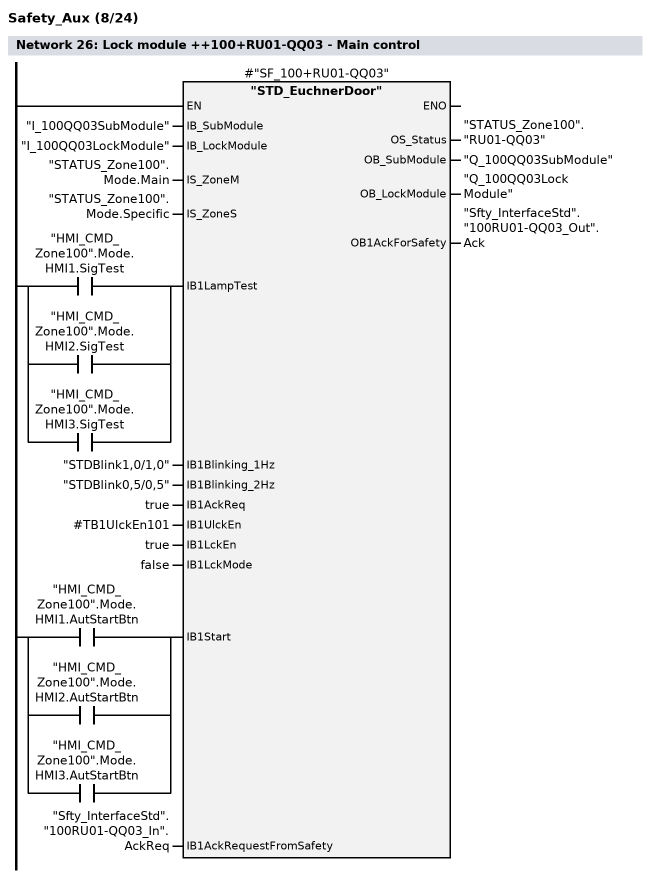
   RUNG wire#powerrail
      #"SF_100+RU01-QQ03"(IB1LampTest := wire#w1, IB1Start := wire#w2, IB_SubModule := "I_100QQ03SubModule", IB_LockModule := "I_100QQ03LockModule", IS_ZoneM := "STATUS_Zone100".Mode.Main, IS_ZoneS := "STATUS_Zone100".Mode.Specific, IB1Blinking_1Hz := "STDBlink1,0/1,0", IB1Blinking_2Hz := "STDBlink0,5/0,5", IB1AckReq := true, IB1UlckEn := #TB1UlckEn101, IB1LckEn := true, IB1LckMode := false, IB1AckRequestFromSafety := "Sfty_InterfaceStd"."100RU01-QQ03_In".AckReq, OS_Status => "STATUS_Zone100"."RU01-QQ03", OB_SubModule => "Q_100QQ03SubModule", OB_LockModule => "Q_100QQ03LockModule", OB1AckForSafety => "Sfty_InterfaceStd"."100RU01-QQ03_Out".Ack)
   END_RUNG
   RUNG wire#powerrail
      Contact( "HMI_CMD_Zone100".Mode.HMI1.SigTest )
   END_RUNG wire#w1
   RUNG wire#powerrail
      Contact( "HMI_CMD_Zone100".Mode.HMI2.SigTest )
   END_RUNG wire#w1
   RUNG wire#powerrail
      Contact( "HMI_CMD_Zone100".Mode.HMI3.SigTest )
   END_RUNG wire#w1
   RUNG wire#powerrail
      Contact( "HMI_CMD_Zone100".Mode.HMI1.AutStartBtn )
   END_RUNG wire#w2
   RUNG wire#powerrail
      Contact( "HMI_CMD_Zone100".Mode.HMI2.AutStartBtn )
   END_RUNG wire#w2
   RUNG wire#powerrail
      Contact( "HMI_CMD_Zone100".Mode.HMI3.AutStartBtn )
   END_RUNG wire#w2
   // the same network as SCL:
   #"SF_100+RU01-QQ03"(IB_SubModule := "I_100QQ03SubModule",   // "STD_EuchnerDoor"
                       IB_LockModule := "I_100QQ03LockModule",
                       IS_ZoneM := "STATUS_Zone100".Mode.Main,
                       IS_ZoneS := "STATUS_Zone100".Mode.Specific,
                       IB1LampTest := "HMI_CMD_Zone100".Mode.HMI1.SigTest OR "HMI_CMD_Zone100".Mode.HMI2.SigTest OR "HMI_CMD_Zone100".Mode.HMI3.SigTest,
                       IB1Blinking_1Hz := "STDBlink1,0/1,0",
                       IB1Blinking_2Hz := "STDBlink0,5/0,5",
                       IB1AckReq := true,
                       IB1UlckEn := #TB1UlckEn101,
                       IB1LckEn := true,
                       IB1LckMode := false,
                       IB1Start := "HMI_CMD_Zone100".Mode.HMI1.AutStartBtn OR "HMI_CMD_Zone100".Mode.HMI2.AutStartBtn OR "HMI_CMD_Zone100".Mode.HMI3.AutStartBtn,
                       IB1AckRequestFromSafety := "Sfty_InterfaceStd"."100RU01-QQ03_In".AckReq,
                       OS_Status => "STATUS_Zone100"."RU01-QQ03",
                       OB_SubModule => "Q_100QQ03SubModule",
                       OB_LockModule => "Q_100QQ03LockModule",
                       OB1AckForSafety => "Sfty_InterfaceStd"."100RU01-QQ03_Out".Ack);
END_REGION

REGION Network 27: Lock module ++100+RU01-QQ04 - Main control
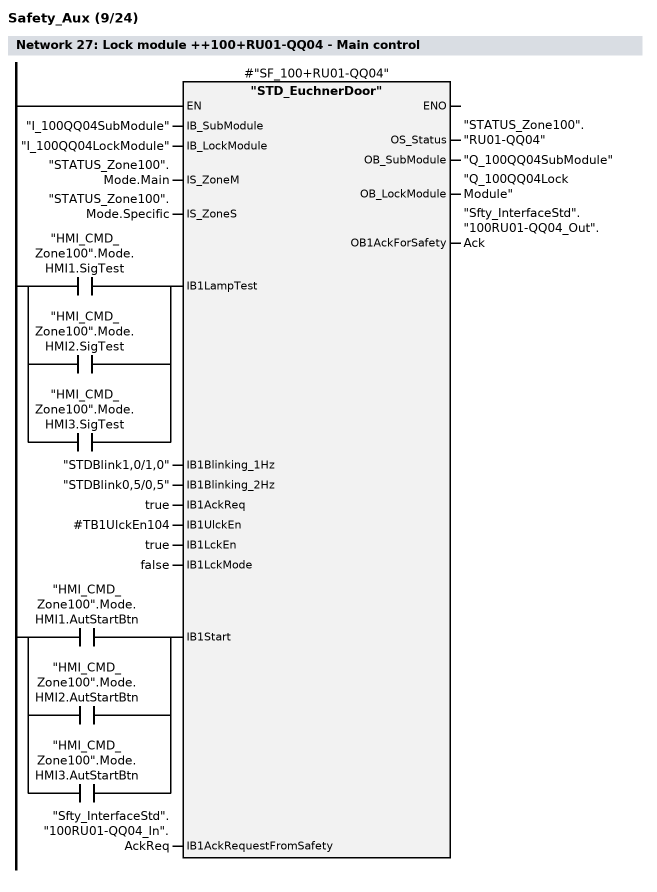
   RUNG wire#powerrail
      #"SF_100+RU01-QQ04"(IB1LampTest := wire#w1, IB1Start := wire#w2, IB_SubModule := "I_100QQ04SubModule", IB_LockModule := "I_100QQ04LockModule", IS_ZoneM := "STATUS_Zone100".Mode.Main, IS_ZoneS := "STATUS_Zone100".Mode.Specific, IB1Blinking_1Hz := "STDBlink1,0/1,0", IB1Blinking_2Hz := "STDBlink0,5/0,5", IB1AckReq := true, IB1UlckEn := #TB1UlckEn104, IB1LckEn := true, IB1LckMode := false, IB1AckRequestFromSafety := "Sfty_InterfaceStd"."100RU01-QQ04_In".AckReq, OS_Status => "STATUS_Zone100"."RU01-QQ04", OB_SubModule => "Q_100QQ04SubModule", OB_LockModule => "Q_100QQ04LockModule", OB1AckForSafety => "Sfty_InterfaceStd"."100RU01-QQ04_Out".Ack)
   END_RUNG
   RUNG wire#powerrail
      Contact( "HMI_CMD_Zone100".Mode.HMI1.SigTest )
   END_RUNG wire#w1
   RUNG wire#powerrail
      Contact( "HMI_CMD_Zone100".Mode.HMI2.SigTest )
   END_RUNG wire#w1
   RUNG wire#powerrail
      Contact( "HMI_CMD_Zone100".Mode.HMI3.SigTest )
   END_RUNG wire#w1
   RUNG wire#powerrail
      Contact( "HMI_CMD_Zone100".Mode.HMI1.AutStartBtn )
   END_RUNG wire#w2
   RUNG wire#powerrail
      Contact( "HMI_CMD_Zone100".Mode.HMI2.AutStartBtn )
   END_RUNG wire#w2
   RUNG wire#powerrail
      Contact( "HMI_CMD_Zone100".Mode.HMI3.AutStartBtn )
   END_RUNG wire#w2
   // the same network as SCL:
   #"SF_100+RU01-QQ04"(IB_SubModule := "I_100QQ04SubModule",   // "STD_EuchnerDoor"
                       IB_LockModule := "I_100QQ04LockModule",
                       IS_ZoneM := "STATUS_Zone100".Mode.Main,
                       IS_ZoneS := "STATUS_Zone100".Mode.Specific,
                       IB1LampTest := "HMI_CMD_Zone100".Mode.HMI1.SigTest OR "HMI_CMD_Zone100".Mode.HMI2.SigTest OR "HMI_CMD_Zone100".Mode.HMI3.SigTest,
                       IB1Blinking_1Hz := "STDBlink1,0/1,0",
                       IB1Blinking_2Hz := "STDBlink0,5/0,5",
                       IB1AckReq := true,
                       IB1UlckEn := #TB1UlckEn104,
                       IB1LckEn := true,
                       IB1LckMode := false,
                       IB1Start := "HMI_CMD_Zone100".Mode.HMI1.AutStartBtn OR "HMI_CMD_Zone100".Mode.HMI2.AutStartBtn OR "HMI_CMD_Zone100".Mode.HMI3.AutStartBtn,
                       IB1AckRequestFromSafety := "Sfty_InterfaceStd"."100RU01-QQ04_In".AckReq,
                       OS_Status => "STATUS_Zone100"."RU01-QQ04",
                       OB_SubModule => "Q_100QQ04SubModule",
                       OB_LockModule => "Q_100QQ04LockModule",
                       OB1AckForSafety => "Sfty_InterfaceStd"."100RU01-QQ04_Out".Ack);
END_REGION

REGION Network 28: Lock module ++100+RU01-QQ05 - Main control
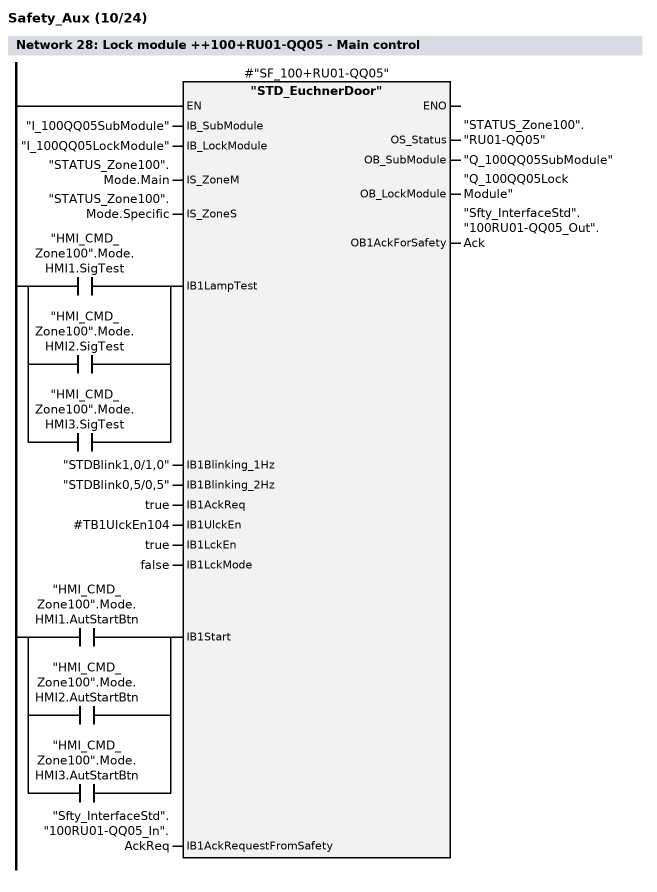
   RUNG wire#powerrail
      #"SF_100+RU01-QQ05"(IB1LampTest := wire#w1, IB1Start := wire#w2, IB_SubModule := "I_100QQ05SubModule", IB_LockModule := "I_100QQ05LockModule", IS_ZoneM := "STATUS_Zone100".Mode.Main, IS_ZoneS := "STATUS_Zone100".Mode.Specific, IB1Blinking_1Hz := "STDBlink1,0/1,0", IB1Blinking_2Hz := "STDBlink0,5/0,5", IB1AckReq := true, IB1UlckEn := #TB1UlckEn104, IB1LckEn := true, IB1LckMode := false, IB1AckRequestFromSafety := "Sfty_InterfaceStd"."100RU01-QQ05_In".AckReq, OS_Status => "STATUS_Zone100"."RU01-QQ05", OB_SubModule => "Q_100QQ05SubModule", OB_LockModule => "Q_100QQ05LockModule", OB1AckForSafety => "Sfty_InterfaceStd"."100RU01-QQ05_Out".Ack)
   END_RUNG
   RUNG wire#powerrail
      Contact( "HMI_CMD_Zone100".Mode.HMI1.SigTest )
   END_RUNG wire#w1
   RUNG wire#powerrail
      Contact( "HMI_CMD_Zone100".Mode.HMI2.SigTest )
   END_RUNG wire#w1
   RUNG wire#powerrail
      Contact( "HMI_CMD_Zone100".Mode.HMI3.SigTest )
   END_RUNG wire#w1
   RUNG wire#powerrail
      Contact( "HMI_CMD_Zone100".Mode.HMI1.AutStartBtn )
   END_RUNG wire#w2
   RUNG wire#powerrail
      Contact( "HMI_CMD_Zone100".Mode.HMI2.AutStartBtn )
   END_RUNG wire#w2
   RUNG wire#powerrail
      Contact( "HMI_CMD_Zone100".Mode.HMI3.AutStartBtn )
   END_RUNG wire#w2
   // the same network as SCL:
   #"SF_100+RU01-QQ05"(IB_SubModule := "I_100QQ05SubModule",   // "STD_EuchnerDoor"
                       IB_LockModule := "I_100QQ05LockModule",
                       IS_ZoneM := "STATUS_Zone100".Mode.Main,
                       IS_ZoneS := "STATUS_Zone100".Mode.Specific,
                       IB1LampTest := "HMI_CMD_Zone100".Mode.HMI1.SigTest OR "HMI_CMD_Zone100".Mode.HMI2.SigTest OR "HMI_CMD_Zone100".Mode.HMI3.SigTest,
                       IB1Blinking_1Hz := "STDBlink1,0/1,0",
                       IB1Blinking_2Hz := "STDBlink0,5/0,5",
                       IB1AckReq := true,
                       IB1UlckEn := #TB1UlckEn104,
                       IB1LckEn := true,
                       IB1LckMode := false,
                       IB1Start := "HMI_CMD_Zone100".Mode.HMI1.AutStartBtn OR "HMI_CMD_Zone100".Mode.HMI2.AutStartBtn OR "HMI_CMD_Zone100".Mode.HMI3.AutStartBtn,
                       IB1AckRequestFromSafety := "Sfty_InterfaceStd"."100RU01-QQ05_In".AckReq,
                       OS_Status => "STATUS_Zone100"."RU01-QQ05",
                       OB_SubModule => "Q_100QQ05SubModule",
                       OB_LockModule => "Q_100QQ05LockModule",
                       OB1AckForSafety => "Sfty_InterfaceStd"."100RU01-QQ05_Out".Ack);
END_REGION

REGION Network 29: Lock module ++100+RU01-QQ06 - Main control
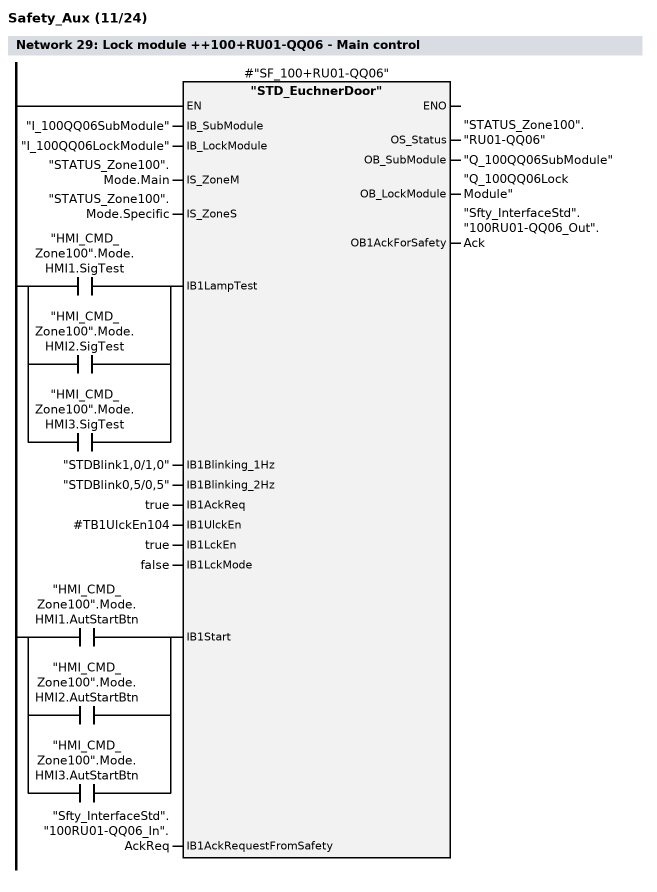
   RUNG wire#powerrail
      #"SF_100+RU01-QQ06"(IB1LampTest := wire#w1, IB1Start := wire#w2, IB_SubModule := "I_100QQ06SubModule", IB_LockModule := "I_100QQ06LockModule", IS_ZoneM := "STATUS_Zone100".Mode.Main, IS_ZoneS := "STATUS_Zone100".Mode.Specific, IB1Blinking_1Hz := "STDBlink1,0/1,0", IB1Blinking_2Hz := "STDBlink0,5/0,5", IB1AckReq := true, IB1UlckEn := #TB1UlckEn104, IB1LckEn := true, IB1LckMode := false, IB1AckRequestFromSafety := "Sfty_InterfaceStd"."100RU01-QQ06_In".AckReq, OS_Status => "STATUS_Zone100"."RU01-QQ06", OB_SubModule => "Q_100QQ06SubModule", OB_LockModule => "Q_100QQ06LockModule", OB1AckForSafety => "Sfty_InterfaceStd"."100RU01-QQ06_Out".Ack)
   END_RUNG
   RUNG wire#powerrail
      Contact( "HMI_CMD_Zone100".Mode.HMI1.SigTest )
   END_RUNG wire#w1
   RUNG wire#powerrail
      Contact( "HMI_CMD_Zone100".Mode.HMI2.SigTest )
   END_RUNG wire#w1
   RUNG wire#powerrail
      Contact( "HMI_CMD_Zone100".Mode.HMI3.SigTest )
   END_RUNG wire#w1
   RUNG wire#powerrail
      Contact( "HMI_CMD_Zone100".Mode.HMI1.AutStartBtn )
   END_RUNG wire#w2
   RUNG wire#powerrail
      Contact( "HMI_CMD_Zone100".Mode.HMI2.AutStartBtn )
   END_RUNG wire#w2
   RUNG wire#powerrail
      Contact( "HMI_CMD_Zone100".Mode.HMI3.AutStartBtn )
   END_RUNG wire#w2
   // the same network as SCL:
   #"SF_100+RU01-QQ06"(IB_SubModule := "I_100QQ06SubModule",   // "STD_EuchnerDoor"
                       IB_LockModule := "I_100QQ06LockModule",
                       IS_ZoneM := "STATUS_Zone100".Mode.Main,
                       IS_ZoneS := "STATUS_Zone100".Mode.Specific,
                       IB1LampTest := "HMI_CMD_Zone100".Mode.HMI1.SigTest OR "HMI_CMD_Zone100".Mode.HMI2.SigTest OR "HMI_CMD_Zone100".Mode.HMI3.SigTest,
                       IB1Blinking_1Hz := "STDBlink1,0/1,0",
                       IB1Blinking_2Hz := "STDBlink0,5/0,5",
                       IB1AckReq := true,
                       IB1UlckEn := #TB1UlckEn104,
                       IB1LckEn := true,
                       IB1LckMode := false,
                       IB1Start := "HMI_CMD_Zone100".Mode.HMI1.AutStartBtn OR "HMI_CMD_Zone100".Mode.HMI2.AutStartBtn OR "HMI_CMD_Zone100".Mode.HMI3.AutStartBtn,
                       IB1AckRequestFromSafety := "Sfty_InterfaceStd"."100RU01-QQ06_In".AckReq,
                       OS_Status => "STATUS_Zone100"."RU01-QQ06",
                       OB_SubModule => "Q_100QQ06SubModule",
                       OB_LockModule => "Q_100QQ06LockModule",
                       OB1AckForSafety => "Sfty_InterfaceStd"."100RU01-QQ06_Out".Ack);
END_REGION

REGION Network 30: Lock module ++100+RU01-QQ07 - Main control
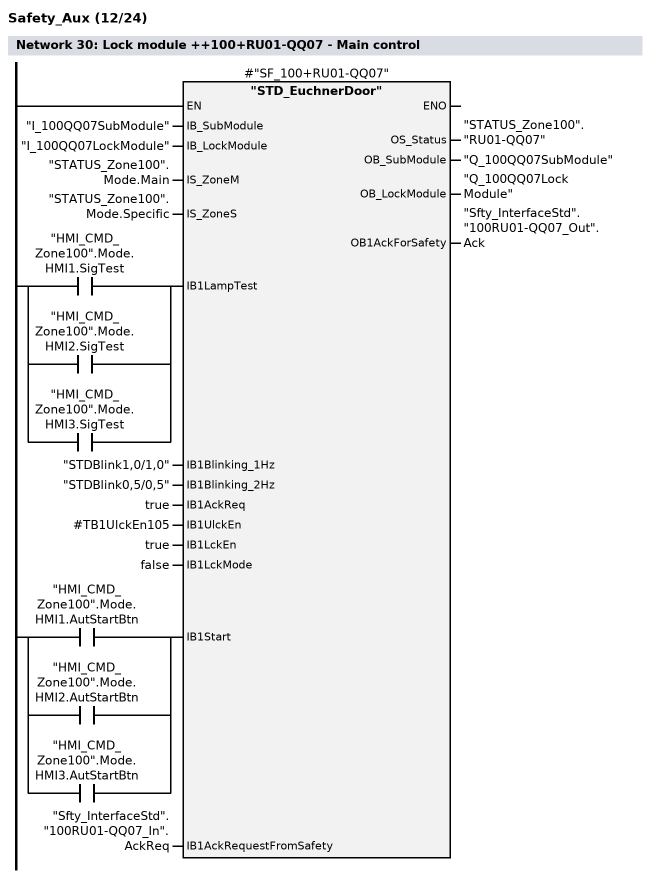
   RUNG wire#powerrail
      #"SF_100+RU01-QQ07"(IB1LampTest := wire#w1, IB1Start := wire#w2, IB_SubModule := "I_100QQ07SubModule", IB_LockModule := "I_100QQ07LockModule", IS_ZoneM := "STATUS_Zone100".Mode.Main, IS_ZoneS := "STATUS_Zone100".Mode.Specific, IB1Blinking_1Hz := "STDBlink1,0/1,0", IB1Blinking_2Hz := "STDBlink0,5/0,5", IB1AckReq := true, IB1UlckEn := #TB1UlckEn105, IB1LckEn := true, IB1LckMode := false, IB1AckRequestFromSafety := "Sfty_InterfaceStd"."100RU01-QQ07_In".AckReq, OS_Status => "STATUS_Zone100"."RU01-QQ07", OB_SubModule => "Q_100QQ07SubModule", OB_LockModule => "Q_100QQ07LockModule", OB1AckForSafety => "Sfty_InterfaceStd"."100RU01-QQ07_Out".Ack)
   END_RUNG
   RUNG wire#powerrail
      Contact( "HMI_CMD_Zone100".Mode.HMI1.SigTest )
   END_RUNG wire#w1
   RUNG wire#powerrail
      Contact( "HMI_CMD_Zone100".Mode.HMI2.SigTest )
   END_RUNG wire#w1
   RUNG wire#powerrail
      Contact( "HMI_CMD_Zone100".Mode.HMI3.SigTest )
   END_RUNG wire#w1
   RUNG wire#powerrail
      Contact( "HMI_CMD_Zone100".Mode.HMI1.AutStartBtn )
   END_RUNG wire#w2
   RUNG wire#powerrail
      Contact( "HMI_CMD_Zone100".Mode.HMI2.AutStartBtn )
   END_RUNG wire#w2
   RUNG wire#powerrail
      Contact( "HMI_CMD_Zone100".Mode.HMI3.AutStartBtn )
   END_RUNG wire#w2
   // the same network as SCL:
   #"SF_100+RU01-QQ07"(IB_SubModule := "I_100QQ07SubModule",   // "STD_EuchnerDoor"
                       IB_LockModule := "I_100QQ07LockModule",
                       IS_ZoneM := "STATUS_Zone100".Mode.Main,
                       IS_ZoneS := "STATUS_Zone100".Mode.Specific,
                       IB1LampTest := "HMI_CMD_Zone100".Mode.HMI1.SigTest OR "HMI_CMD_Zone100".Mode.HMI2.SigTest OR "HMI_CMD_Zone100".Mode.HMI3.SigTest,
                       IB1Blinking_1Hz := "STDBlink1,0/1,0",
                       IB1Blinking_2Hz := "STDBlink0,5/0,5",
                       IB1AckReq := true,
                       IB1UlckEn := #TB1UlckEn105,
                       IB1LckEn := true,
                       IB1LckMode := false,
                       IB1Start := "HMI_CMD_Zone100".Mode.HMI1.AutStartBtn OR "HMI_CMD_Zone100".Mode.HMI2.AutStartBtn OR "HMI_CMD_Zone100".Mode.HMI3.AutStartBtn,
                       IB1AckRequestFromSafety := "Sfty_InterfaceStd"."100RU01-QQ07_In".AckReq,
                       OS_Status => "STATUS_Zone100"."RU01-QQ07",
                       OB_SubModule => "Q_100QQ07SubModule",
                       OB_LockModule => "Q_100QQ07LockModule",
                       OB1AckForSafety => "Sfty_InterfaceStd"."100RU01-QQ07_Out".Ack);
END_REGION

REGION Network 31: Lock module ++100+RU01-QQ08 - Main control
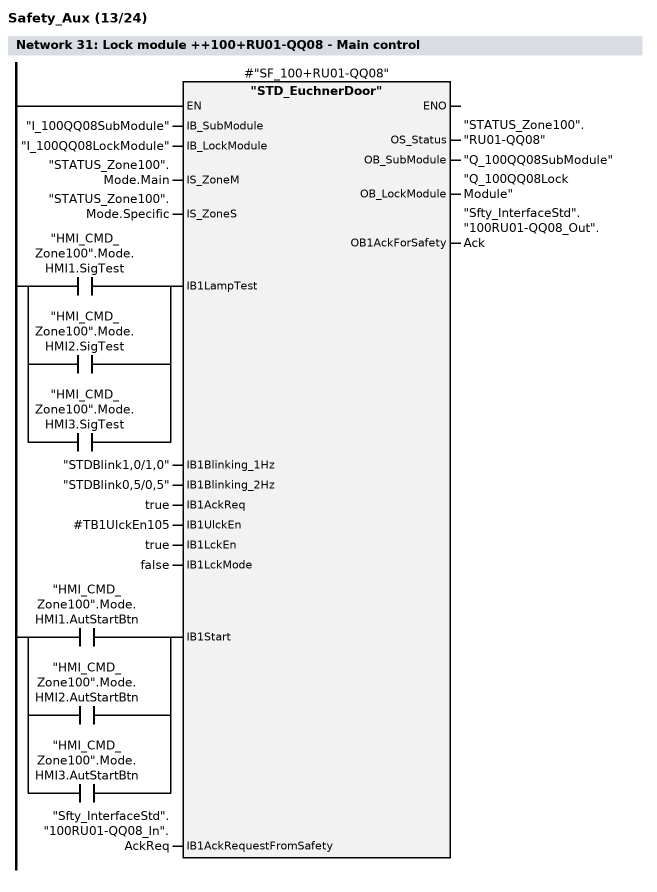
   RUNG wire#powerrail
      #"SF_100+RU01-QQ08"(IB1LampTest := wire#w1, IB1Start := wire#w2, IB_SubModule := "I_100QQ08SubModule", IB_LockModule := "I_100QQ08LockModule", IS_ZoneM := "STATUS_Zone100".Mode.Main, IS_ZoneS := "STATUS_Zone100".Mode.Specific, IB1Blinking_1Hz := "STDBlink1,0/1,0", IB1Blinking_2Hz := "STDBlink0,5/0,5", IB1AckReq := true, IB1UlckEn := #TB1UlckEn105, IB1LckEn := true, IB1LckMode := false, IB1AckRequestFromSafety := "Sfty_InterfaceStd"."100RU01-QQ08_In".AckReq, OS_Status => "STATUS_Zone100"."RU01-QQ08", OB_SubModule => "Q_100QQ08SubModule", OB_LockModule => "Q_100QQ08LockModule", OB1AckForSafety => "Sfty_InterfaceStd"."100RU01-QQ08_Out".Ack)
   END_RUNG
   RUNG wire#powerrail
      Contact( "HMI_CMD_Zone100".Mode.HMI1.SigTest )
   END_RUNG wire#w1
   RUNG wire#powerrail
      Contact( "HMI_CMD_Zone100".Mode.HMI2.SigTest )
   END_RUNG wire#w1
   RUNG wire#powerrail
      Contact( "HMI_CMD_Zone100".Mode.HMI3.SigTest )
   END_RUNG wire#w1
   RUNG wire#powerrail
      Contact( "HMI_CMD_Zone100".Mode.HMI1.AutStartBtn )
   END_RUNG wire#w2
   RUNG wire#powerrail
      Contact( "HMI_CMD_Zone100".Mode.HMI2.AutStartBtn )
   END_RUNG wire#w2
   RUNG wire#powerrail
      Contact( "HMI_CMD_Zone100".Mode.HMI3.AutStartBtn )
   END_RUNG wire#w2
   // the same network as SCL:
   #"SF_100+RU01-QQ08"(IB_SubModule := "I_100QQ08SubModule",   // "STD_EuchnerDoor"
                       IB_LockModule := "I_100QQ08LockModule",
                       IS_ZoneM := "STATUS_Zone100".Mode.Main,
                       IS_ZoneS := "STATUS_Zone100".Mode.Specific,
                       IB1LampTest := "HMI_CMD_Zone100".Mode.HMI1.SigTest OR "HMI_CMD_Zone100".Mode.HMI2.SigTest OR "HMI_CMD_Zone100".Mode.HMI3.SigTest,
                       IB1Blinking_1Hz := "STDBlink1,0/1,0",
                       IB1Blinking_2Hz := "STDBlink0,5/0,5",
                       IB1AckReq := true,
                       IB1UlckEn := #TB1UlckEn105,
                       IB1LckEn := true,
                       IB1LckMode := false,
                       IB1Start := "HMI_CMD_Zone100".Mode.HMI1.AutStartBtn OR "HMI_CMD_Zone100".Mode.HMI2.AutStartBtn OR "HMI_CMD_Zone100".Mode.HMI3.AutStartBtn,
                       IB1AckRequestFromSafety := "Sfty_InterfaceStd"."100RU01-QQ08_In".AckReq,
                       OS_Status => "STATUS_Zone100"."RU01-QQ08",
                       OB_SubModule => "Q_100QQ08SubModule",
                       OB_LockModule => "Q_100QQ08LockModule",
                       OB1AckForSafety => "Sfty_InterfaceStd"."100RU01-QQ08_Out".Ack);
END_REGION

REGION Network 32: Lock module ++200+RU01-QQ01 - Main control
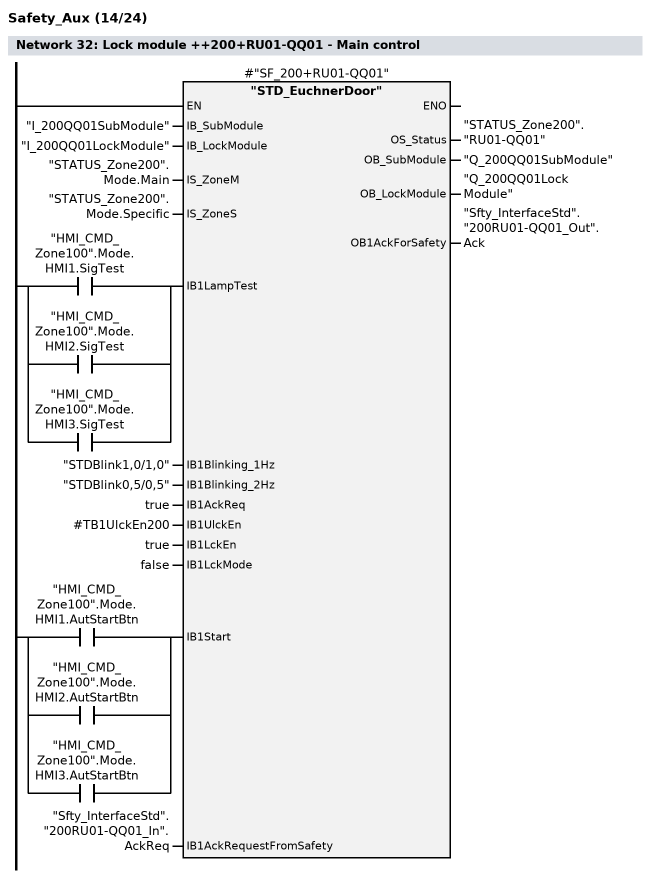
   RUNG wire#powerrail
      #"SF_200+RU01-QQ01"(IB1LampTest := wire#w1, IB1Start := wire#w2, IB_SubModule := "I_200QQ01SubModule", IB_LockModule := "I_200QQ01LockModule", IS_ZoneM := "STATUS_Zone200".Mode.Main, IS_ZoneS := "STATUS_Zone200".Mode.Specific, IB1Blinking_1Hz := "STDBlink1,0/1,0", IB1Blinking_2Hz := "STDBlink0,5/0,5", IB1AckReq := true, IB1UlckEn := #TB1UlckEn200, IB1LckEn := true, IB1LckMode := false, IB1AckRequestFromSafety := "Sfty_InterfaceStd"."200RU01-QQ01_In".AckReq, OS_Status => "STATUS_Zone200"."RU01-QQ01", OB_SubModule => "Q_200QQ01SubModule", OB_LockModule => "Q_200QQ01LockModule", OB1AckForSafety => "Sfty_InterfaceStd"."200RU01-QQ01_Out".Ack)
   END_RUNG
   RUNG wire#powerrail
      Contact( "HMI_CMD_Zone100".Mode.HMI1.SigTest )
   END_RUNG wire#w1
   RUNG wire#powerrail
      Contact( "HMI_CMD_Zone100".Mode.HMI2.SigTest )
   END_RUNG wire#w1
   RUNG wire#powerrail
      Contact( "HMI_CMD_Zone100".Mode.HMI3.SigTest )
   END_RUNG wire#w1
   RUNG wire#powerrail
      Contact( "HMI_CMD_Zone100".Mode.HMI1.AutStartBtn )
   END_RUNG wire#w2
   RUNG wire#powerrail
      Contact( "HMI_CMD_Zone100".Mode.HMI2.AutStartBtn )
   END_RUNG wire#w2
   RUNG wire#powerrail
      Contact( "HMI_CMD_Zone100".Mode.HMI3.AutStartBtn )
   END_RUNG wire#w2
   // the same network as SCL:
   #"SF_200+RU01-QQ01"(IB_SubModule := "I_200QQ01SubModule",   // "STD_EuchnerDoor"
                       IB_LockModule := "I_200QQ01LockModule",
                       IS_ZoneM := "STATUS_Zone200".Mode.Main,
                       IS_ZoneS := "STATUS_Zone200".Mode.Specific,
                       IB1LampTest := "HMI_CMD_Zone100".Mode.HMI1.SigTest OR "HMI_CMD_Zone100".Mode.HMI2.SigTest OR "HMI_CMD_Zone100".Mode.HMI3.SigTest,
                       IB1Blinking_1Hz := "STDBlink1,0/1,0",
                       IB1Blinking_2Hz := "STDBlink0,5/0,5",
                       IB1AckReq := true,
                       IB1UlckEn := #TB1UlckEn200,
                       IB1LckEn := true,
                       IB1LckMode := false,
                       IB1Start := "HMI_CMD_Zone100".Mode.HMI1.AutStartBtn OR "HMI_CMD_Zone100".Mode.HMI2.AutStartBtn OR "HMI_CMD_Zone100".Mode.HMI3.AutStartBtn,
                       IB1AckRequestFromSafety := "Sfty_InterfaceStd"."200RU01-QQ01_In".AckReq,
                       OS_Status => "STATUS_Zone200"."RU01-QQ01",
                       OB_SubModule => "Q_200QQ01SubModule",
                       OB_LockModule => "Q_200QQ01LockModule",
                       OB1AckForSafety => "Sfty_InterfaceStd"."200RU01-QQ01_Out".Ack);
END_REGION

REGION Network 33: Lock module ++200+RU01-QQ02 - Main control
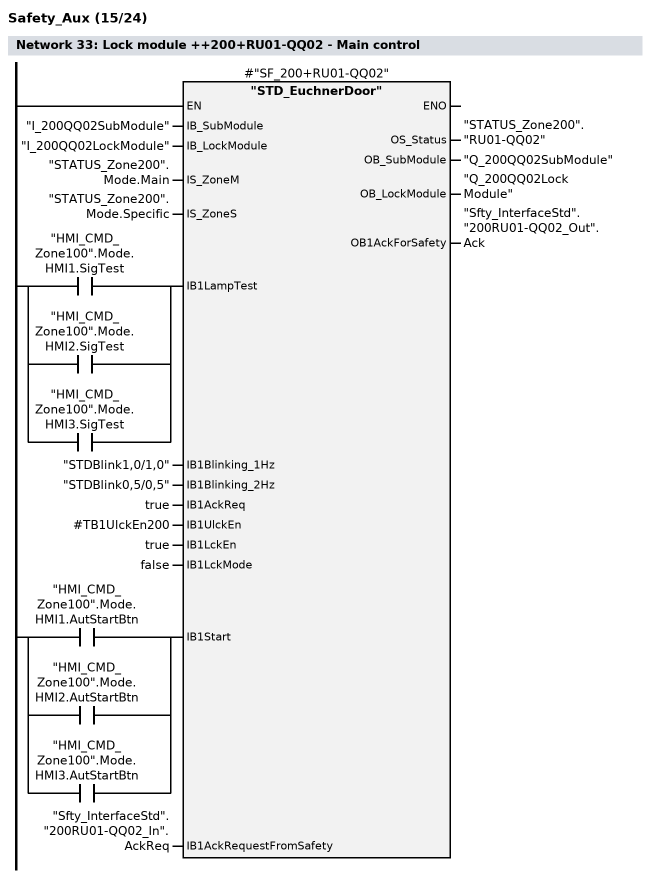
   RUNG wire#powerrail
      #"SF_200+RU01-QQ02"(IB1LampTest := wire#w1, IB1Start := wire#w2, IB_SubModule := "I_200QQ02SubModule", IB_LockModule := "I_200QQ02LockModule", IS_ZoneM := "STATUS_Zone200".Mode.Main, IS_ZoneS := "STATUS_Zone200".Mode.Specific, IB1Blinking_1Hz := "STDBlink1,0/1,0", IB1Blinking_2Hz := "STDBlink0,5/0,5", IB1AckReq := true, IB1UlckEn := #TB1UlckEn200, IB1LckEn := true, IB1LckMode := false, IB1AckRequestFromSafety := "Sfty_InterfaceStd"."200RU01-QQ02_In".AckReq, OS_Status => "STATUS_Zone200"."RU01-QQ02", OB_SubModule => "Q_200QQ02SubModule", OB_LockModule => "Q_200QQ02LockModule", OB1AckForSafety => "Sfty_InterfaceStd"."200RU01-QQ02_Out".Ack)
   END_RUNG
   RUNG wire#powerrail
      Contact( "HMI_CMD_Zone100".Mode.HMI1.SigTest )
   END_RUNG wire#w1
   RUNG wire#powerrail
      Contact( "HMI_CMD_Zone100".Mode.HMI2.SigTest )
   END_RUNG wire#w1
   RUNG wire#powerrail
      Contact( "HMI_CMD_Zone100".Mode.HMI3.SigTest )
   END_RUNG wire#w1
   RUNG wire#powerrail
      Contact( "HMI_CMD_Zone100".Mode.HMI1.AutStartBtn )
   END_RUNG wire#w2
   RUNG wire#powerrail
      Contact( "HMI_CMD_Zone100".Mode.HMI2.AutStartBtn )
   END_RUNG wire#w2
   RUNG wire#powerrail
      Contact( "HMI_CMD_Zone100".Mode.HMI3.AutStartBtn )
   END_RUNG wire#w2
   // the same network as SCL:
   #"SF_200+RU01-QQ02"(IB_SubModule := "I_200QQ02SubModule",   // "STD_EuchnerDoor"
                       IB_LockModule := "I_200QQ02LockModule",
                       IS_ZoneM := "STATUS_Zone200".Mode.Main,
                       IS_ZoneS := "STATUS_Zone200".Mode.Specific,
                       IB1LampTest := "HMI_CMD_Zone100".Mode.HMI1.SigTest OR "HMI_CMD_Zone100".Mode.HMI2.SigTest OR "HMI_CMD_Zone100".Mode.HMI3.SigTest,
                       IB1Blinking_1Hz := "STDBlink1,0/1,0",
                       IB1Blinking_2Hz := "STDBlink0,5/0,5",
                       IB1AckReq := true,
                       IB1UlckEn := #TB1UlckEn200,
                       IB1LckEn := true,
                       IB1LckMode := false,
                       IB1Start := "HMI_CMD_Zone100".Mode.HMI1.AutStartBtn OR "HMI_CMD_Zone100".Mode.HMI2.AutStartBtn OR "HMI_CMD_Zone100".Mode.HMI3.AutStartBtn,
                       IB1AckRequestFromSafety := "Sfty_InterfaceStd"."200RU01-QQ02_In".AckReq,
                       OS_Status => "STATUS_Zone200"."RU01-QQ02",
                       OB_SubModule => "Q_200QQ02SubModule",
                       OB_LockModule => "Q_200QQ02LockModule",
                       OB1AckForSafety => "Sfty_InterfaceStd"."200RU01-QQ02_Out".Ack);
END_REGION

REGION Network 34: Lock module ++200+RU01-QQ03 - Main control
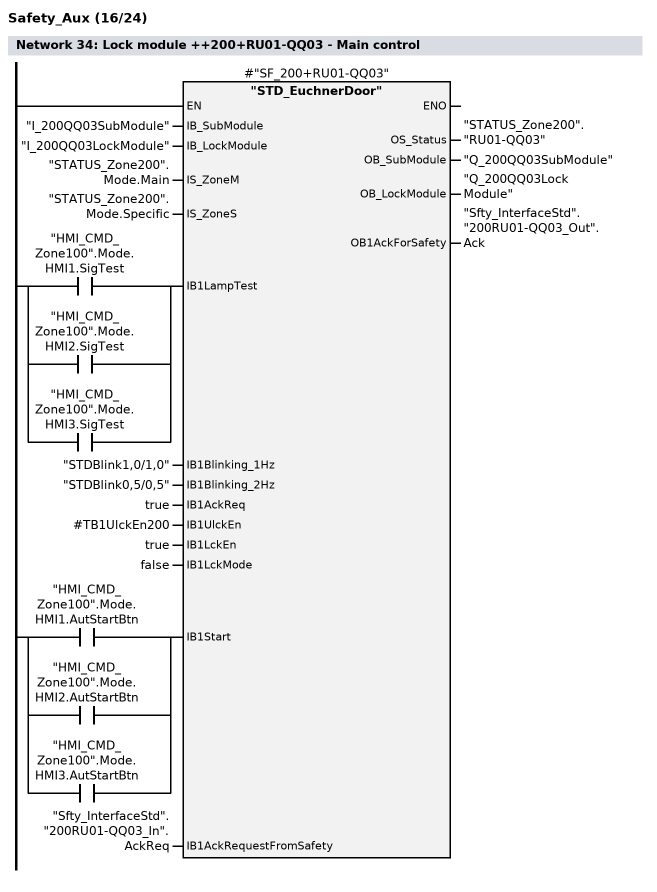
   RUNG wire#powerrail
      #"SF_200+RU01-QQ03"(IB1LampTest := wire#w1, IB1Start := wire#w2, IB_SubModule := "I_200QQ03SubModule", IB_LockModule := "I_200QQ03LockModule", IS_ZoneM := "STATUS_Zone200".Mode.Main, IS_ZoneS := "STATUS_Zone200".Mode.Specific, IB1Blinking_1Hz := "STDBlink1,0/1,0", IB1Blinking_2Hz := "STDBlink0,5/0,5", IB1AckReq := true, IB1UlckEn := #TB1UlckEn200, IB1LckEn := true, IB1LckMode := false, IB1AckRequestFromSafety := "Sfty_InterfaceStd"."200RU01-QQ03_In".AckReq, OS_Status => "STATUS_Zone200"."RU01-QQ03", OB_SubModule => "Q_200QQ03SubModule", OB_LockModule => "Q_200QQ03LockModule", OB1AckForSafety => "Sfty_InterfaceStd"."200RU01-QQ03_Out".Ack)
   END_RUNG
   RUNG wire#powerrail
      Contact( "HMI_CMD_Zone100".Mode.HMI1.SigTest )
   END_RUNG wire#w1
   RUNG wire#powerrail
      Contact( "HMI_CMD_Zone100".Mode.HMI2.SigTest )
   END_RUNG wire#w1
   RUNG wire#powerrail
      Contact( "HMI_CMD_Zone100".Mode.HMI3.SigTest )
   END_RUNG wire#w1
   RUNG wire#powerrail
      Contact( "HMI_CMD_Zone100".Mode.HMI1.AutStartBtn )
   END_RUNG wire#w2
   RUNG wire#powerrail
      Contact( "HMI_CMD_Zone100".Mode.HMI2.AutStartBtn )
   END_RUNG wire#w2
   RUNG wire#powerrail
      Contact( "HMI_CMD_Zone100".Mode.HMI3.AutStartBtn )
   END_RUNG wire#w2
   // the same network as SCL:
   #"SF_200+RU01-QQ03"(IB_SubModule := "I_200QQ03SubModule",   // "STD_EuchnerDoor"
                       IB_LockModule := "I_200QQ03LockModule",
                       IS_ZoneM := "STATUS_Zone200".Mode.Main,
                       IS_ZoneS := "STATUS_Zone200".Mode.Specific,
                       IB1LampTest := "HMI_CMD_Zone100".Mode.HMI1.SigTest OR "HMI_CMD_Zone100".Mode.HMI2.SigTest OR "HMI_CMD_Zone100".Mode.HMI3.SigTest,
                       IB1Blinking_1Hz := "STDBlink1,0/1,0",
                       IB1Blinking_2Hz := "STDBlink0,5/0,5",
                       IB1AckReq := true,
                       IB1UlckEn := #TB1UlckEn200,
                       IB1LckEn := true,
                       IB1LckMode := false,
                       IB1Start := "HMI_CMD_Zone100".Mode.HMI1.AutStartBtn OR "HMI_CMD_Zone100".Mode.HMI2.AutStartBtn OR "HMI_CMD_Zone100".Mode.HMI3.AutStartBtn,
                       IB1AckRequestFromSafety := "Sfty_InterfaceStd"."200RU01-QQ03_In".AckReq,
                       OS_Status => "STATUS_Zone200"."RU01-QQ03",
                       OB_SubModule => "Q_200QQ03SubModule",
                       OB_LockModule => "Q_200QQ03LockModule",
                       OB1AckForSafety => "Sfty_InterfaceStd"."200RU01-QQ03_Out".Ack);
END_REGION

REGION Network 35: Lock module ++200+RU01-QQ04 - Main control
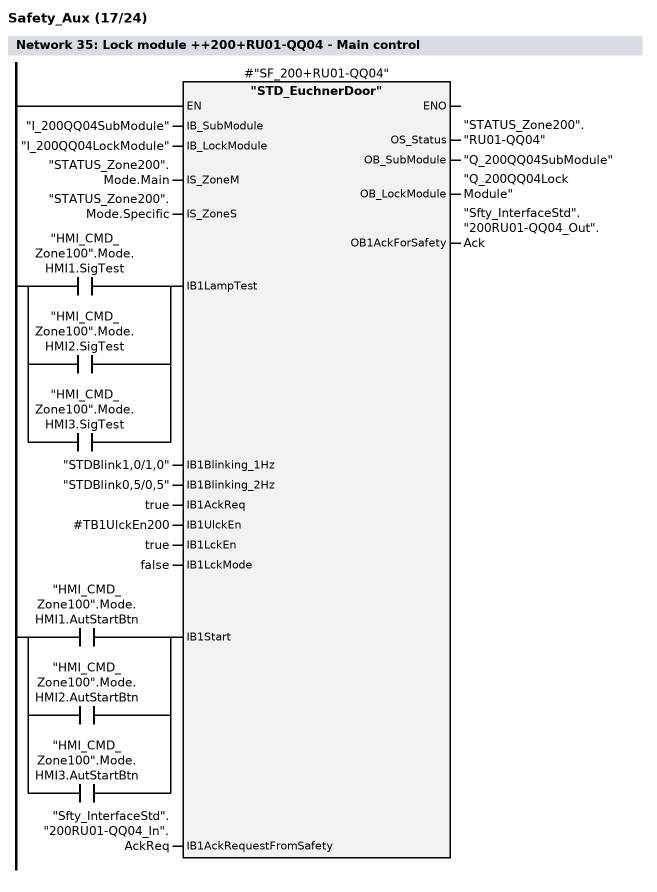
   RUNG wire#powerrail
      #"SF_200+RU01-QQ04"(IB1LampTest := wire#w1, IB1Start := wire#w2, IB_SubModule := "I_200QQ04SubModule", IB_LockModule := "I_200QQ04LockModule", IS_ZoneM := "STATUS_Zone200".Mode.Main, IS_ZoneS := "STATUS_Zone200".Mode.Specific, IB1Blinking_1Hz := "STDBlink1,0/1,0", IB1Blinking_2Hz := "STDBlink0,5/0,5", IB1AckReq := true, IB1UlckEn := #TB1UlckEn200, IB1LckEn := true, IB1LckMode := false, IB1AckRequestFromSafety := "Sfty_InterfaceStd"."200RU01-QQ04_In".AckReq, OS_Status => "STATUS_Zone200"."RU01-QQ04", OB_SubModule => "Q_200QQ04SubModule", OB_LockModule => "Q_200QQ04LockModule", OB1AckForSafety => "Sfty_InterfaceStd"."200RU01-QQ04_Out".Ack)
   END_RUNG
   RUNG wire#powerrail
      Contact( "HMI_CMD_Zone100".Mode.HMI1.SigTest )
   END_RUNG wire#w1
   RUNG wire#powerrail
      Contact( "HMI_CMD_Zone100".Mode.HMI2.SigTest )
   END_RUNG wire#w1
   RUNG wire#powerrail
      Contact( "HMI_CMD_Zone100".Mode.HMI3.SigTest )
   END_RUNG wire#w1
   RUNG wire#powerrail
      Contact( "HMI_CMD_Zone100".Mode.HMI1.AutStartBtn )
   END_RUNG wire#w2
   RUNG wire#powerrail
      Contact( "HMI_CMD_Zone100".Mode.HMI2.AutStartBtn )
   END_RUNG wire#w2
   RUNG wire#powerrail
      Contact( "HMI_CMD_Zone100".Mode.HMI3.AutStartBtn )
   END_RUNG wire#w2
   // the same network as SCL:
   #"SF_200+RU01-QQ04"(IB_SubModule := "I_200QQ04SubModule",   // "STD_EuchnerDoor"
                       IB_LockModule := "I_200QQ04LockModule",
                       IS_ZoneM := "STATUS_Zone200".Mode.Main,
                       IS_ZoneS := "STATUS_Zone200".Mode.Specific,
                       IB1LampTest := "HMI_CMD_Zone100".Mode.HMI1.SigTest OR "HMI_CMD_Zone100".Mode.HMI2.SigTest OR "HMI_CMD_Zone100".Mode.HMI3.SigTest,
                       IB1Blinking_1Hz := "STDBlink1,0/1,0",
                       IB1Blinking_2Hz := "STDBlink0,5/0,5",
                       IB1AckReq := true,
                       IB1UlckEn := #TB1UlckEn200,
                       IB1LckEn := true,
                       IB1LckMode := false,
                       IB1Start := "HMI_CMD_Zone100".Mode.HMI1.AutStartBtn OR "HMI_CMD_Zone100".Mode.HMI2.AutStartBtn OR "HMI_CMD_Zone100".Mode.HMI3.AutStartBtn,
                       IB1AckRequestFromSafety := "Sfty_InterfaceStd"."200RU01-QQ04_In".AckReq,
                       OS_Status => "STATUS_Zone200"."RU01-QQ04",
                       OB_SubModule => "Q_200QQ04SubModule",
                       OB_LockModule => "Q_200QQ04LockModule",
                       OB1AckForSafety => "Sfty_InterfaceStd"."200RU01-QQ04_Out".Ack);
END_REGION

REGION Network 36: Lock module ++200+RU01-QQ05 - Main control
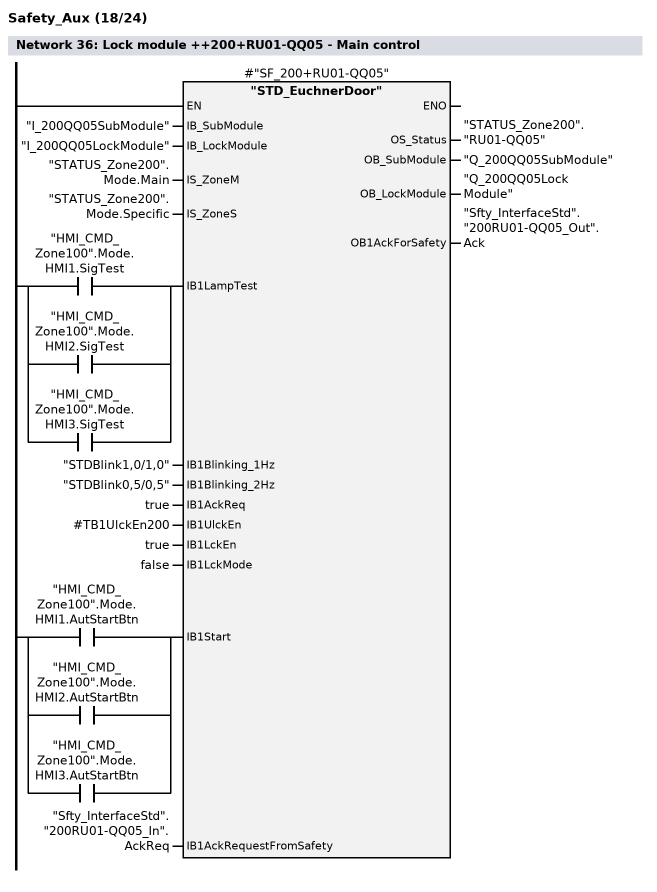
   RUNG wire#powerrail
      #"SF_200+RU01-QQ05"(IB1LampTest := wire#w1, IB1Start := wire#w2, IB_SubModule := "I_200QQ05SubModule", IB_LockModule := "I_200QQ05LockModule", IS_ZoneM := "STATUS_Zone200".Mode.Main, IS_ZoneS := "STATUS_Zone200".Mode.Specific, IB1Blinking_1Hz := "STDBlink1,0/1,0", IB1Blinking_2Hz := "STDBlink0,5/0,5", IB1AckReq := true, IB1UlckEn := #TB1UlckEn200, IB1LckEn := true, IB1LckMode := false, IB1AckRequestFromSafety := "Sfty_InterfaceStd"."200RU01-QQ05_In".AckReq, OS_Status => "STATUS_Zone200"."RU01-QQ05", OB_SubModule => "Q_200QQ05SubModule", OB_LockModule => "Q_200QQ05LockModule", OB1AckForSafety => "Sfty_InterfaceStd"."200RU01-QQ05_Out".Ack)
   END_RUNG
   RUNG wire#powerrail
      Contact( "HMI_CMD_Zone100".Mode.HMI1.SigTest )
   END_RUNG wire#w1
   RUNG wire#powerrail
      Contact( "HMI_CMD_Zone100".Mode.HMI2.SigTest )
   END_RUNG wire#w1
   RUNG wire#powerrail
      Contact( "HMI_CMD_Zone100".Mode.HMI3.SigTest )
   END_RUNG wire#w1
   RUNG wire#powerrail
      Contact( "HMI_CMD_Zone100".Mode.HMI1.AutStartBtn )
   END_RUNG wire#w2
   RUNG wire#powerrail
      Contact( "HMI_CMD_Zone100".Mode.HMI2.AutStartBtn )
   END_RUNG wire#w2
   RUNG wire#powerrail
      Contact( "HMI_CMD_Zone100".Mode.HMI3.AutStartBtn )
   END_RUNG wire#w2
   // the same network as SCL:
   #"SF_200+RU01-QQ05"(IB_SubModule := "I_200QQ05SubModule",   // "STD_EuchnerDoor"
                       IB_LockModule := "I_200QQ05LockModule",
                       IS_ZoneM := "STATUS_Zone200".Mode.Main,
                       IS_ZoneS := "STATUS_Zone200".Mode.Specific,
                       IB1LampTest := "HMI_CMD_Zone100".Mode.HMI1.SigTest OR "HMI_CMD_Zone100".Mode.HMI2.SigTest OR "HMI_CMD_Zone100".Mode.HMI3.SigTest,
                       IB1Blinking_1Hz := "STDBlink1,0/1,0",
                       IB1Blinking_2Hz := "STDBlink0,5/0,5",
                       IB1AckReq := true,
                       IB1UlckEn := #TB1UlckEn200,
                       IB1LckEn := true,
                       IB1LckMode := false,
                       IB1Start := "HMI_CMD_Zone100".Mode.HMI1.AutStartBtn OR "HMI_CMD_Zone100".Mode.HMI2.AutStartBtn OR "HMI_CMD_Zone100".Mode.HMI3.AutStartBtn,
                       IB1AckRequestFromSafety := "Sfty_InterfaceStd"."200RU01-QQ05_In".AckReq,
                       OS_Status => "STATUS_Zone200"."RU01-QQ05",
                       OB_SubModule => "Q_200QQ05SubModule",
                       OB_LockModule => "Q_200QQ05LockModule",
                       OB1AckForSafety => "Sfty_InterfaceStd"."200RU01-QQ05_Out".Ack);
END_REGION

REGION Network 37: *************** Alarms estop suppliers ***************
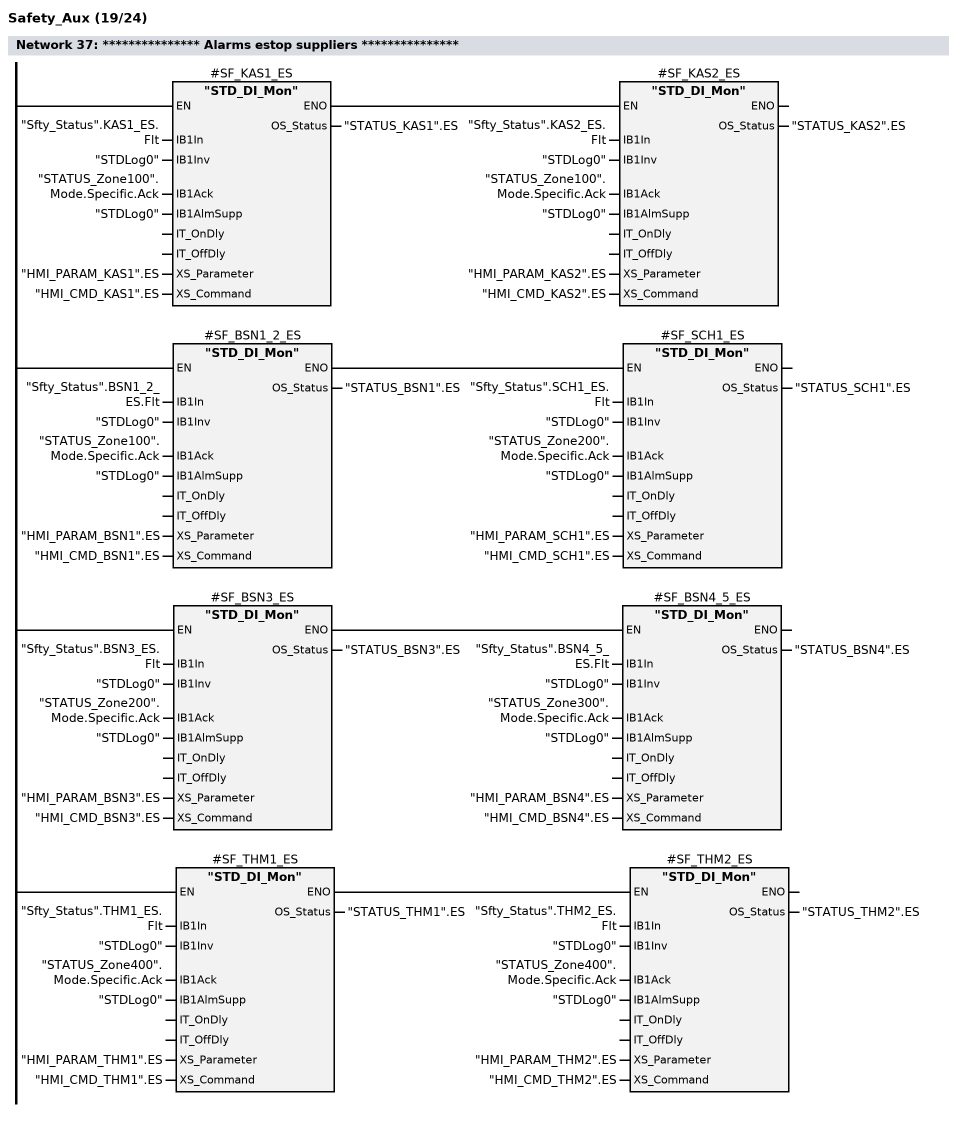
   RUNG wire#powerrail
      #SF_KAS1_ES(IB1In := "Sfty_Status".KAS1_ES.Flt, IB1Inv := "STDLog0", IB1Ack := "STATUS_Zone100".Mode.Specific.Ack, IB1AlmSupp := "STDLog0", IT_OnDly :=, IT_OffDly :=, XS_Parameter := "HMI_PARAM_KAS1".ES, XS_Command := "HMI_CMD_KAS1".ES, OS_Status => "STATUS_KAS1".ES)
      #SF_KAS2_ES(IB1In := "Sfty_Status".KAS2_ES.Flt, IB1Inv := "STDLog0", IB1Ack := "STATUS_Zone100".Mode.Specific.Ack, IB1AlmSupp := "STDLog0", IT_OnDly :=, IT_OffDly :=, XS_Parameter := "HMI_PARAM_KAS2".ES, XS_Command := "HMI_CMD_KAS2".ES, OS_Status => "STATUS_KAS2".ES)
   END_RUNG
   RUNG wire#powerrail
      #SF_BSN1_2_ES(IB1In := "Sfty_Status".BSN1_2_ES.Flt, IB1Inv := "STDLog0", IB1Ack := "STATUS_Zone100".Mode.Specific.Ack, IB1AlmSupp := "STDLog0", IT_OnDly :=, IT_OffDly :=, XS_Parameter := "HMI_PARAM_BSN1".ES, XS_Command := "HMI_CMD_BSN1".ES, OS_Status => "STATUS_BSN1".ES)
      #SF_SCH1_ES(IB1In := "Sfty_Status".SCH1_ES.Flt, IB1Inv := "STDLog0", IB1Ack := "STATUS_Zone200".Mode.Specific.Ack, IB1AlmSupp := "STDLog0", IT_OnDly :=, IT_OffDly :=, XS_Parameter := "HMI_PARAM_SCH1".ES, XS_Command := "HMI_CMD_SCH1".ES, OS_Status => "STATUS_SCH1".ES)
   END_RUNG
   RUNG wire#powerrail
      #SF_BSN3_ES(IB1In := "Sfty_Status".BSN3_ES.Flt, IB1Inv := "STDLog0", IB1Ack := "STATUS_Zone200".Mode.Specific.Ack, IB1AlmSupp := "STDLog0", IT_OnDly :=, IT_OffDly :=, XS_Parameter := "HMI_PARAM_BSN3".ES, XS_Command := "HMI_CMD_BSN3".ES, OS_Status => "STATUS_BSN3".ES)
      #SF_BSN4_5_ES(IB1In := "Sfty_Status".BSN4_5_ES.Flt, IB1Inv := "STDLog0", IB1Ack := "STATUS_Zone300".Mode.Specific.Ack, IB1AlmSupp := "STDLog0", IT_OnDly :=, IT_OffDly :=, XS_Parameter := "HMI_PARAM_BSN4".ES, XS_Command := "HMI_CMD_BSN4".ES, OS_Status => "STATUS_BSN4".ES)
   END_RUNG
   RUNG wire#powerrail
      #SF_THM1_ES(IB1In := "Sfty_Status".THM1_ES.Flt, IB1Inv := "STDLog0", IB1Ack := "STATUS_Zone400".Mode.Specific.Ack, IB1AlmSupp := "STDLog0", IT_OnDly :=, IT_OffDly :=, XS_Parameter := "HMI_PARAM_THM1".ES, XS_Command := "HMI_CMD_THM1".ES, OS_Status => "STATUS_THM1".ES)
      #SF_THM2_ES(IB1In := "Sfty_Status".THM2_ES.Flt, IB1Inv := "STDLog0", IB1Ack := "STATUS_Zone400".Mode.Specific.Ack, IB1AlmSupp := "STDLog0", IT_OnDly :=, IT_OffDly :=, XS_Parameter := "HMI_PARAM_THM2".ES, XS_Command := "HMI_CMD_THM2".ES, OS_Status => "STATUS_THM2".ES)
   END_RUNG
   // the same network as SCL:
   #SF_KAS1_ES(IB1In := "Sfty_Status".KAS1_ES.Flt,   // "STD_DI_Mon"
               IB1Inv := "STDLog0",
               IB1Ack := "STATUS_Zone100".Mode.Specific.Ack,
               IB1AlmSupp := "STDLog0",
               XS_Parameter := "HMI_PARAM_KAS1".ES,
               XS_Command := "HMI_CMD_KAS1".ES,
               OS_Status => "STATUS_KAS1".ES,
               ENO => #_w1);
   IF #_w1 THEN
       #SF_KAS2_ES(IB1In := "Sfty_Status".KAS2_ES.Flt,   // "STD_DI_Mon"
                   IB1Inv := "STDLog0",
                   IB1Ack := "STATUS_Zone100".Mode.Specific.Ack,
                   IB1AlmSupp := "STDLog0",
                   XS_Parameter := "HMI_PARAM_KAS2".ES,
                   XS_Command := "HMI_CMD_KAS2".ES,
                   OS_Status => "STATUS_KAS2".ES);
   END_IF;
   #SF_BSN1_2_ES(IB1In := "Sfty_Status".BSN1_2_ES.Flt,   // "STD_DI_Mon"
                 IB1Inv := "STDLog0",
                 IB1Ack := "STATUS_Zone100".Mode.Specific.Ack,
                 IB1AlmSupp := "STDLog0",
                 XS_Parameter := "HMI_PARAM_BSN1".ES,
                 XS_Command := "HMI_CMD_BSN1".ES,
                 OS_Status => "STATUS_BSN1".ES,
                 ENO => #_w2);
   IF #_w2 THEN
       #SF_SCH1_ES(IB1In := "Sfty_Status".SCH1_ES.Flt,   // "STD_DI_Mon"
                   IB1Inv := "STDLog0",
                   IB1Ack := "STATUS_Zone200".Mode.Specific.Ack,
                   IB1AlmSupp := "STDLog0",
                   XS_Parameter := "HMI_PARAM_SCH1".ES,
                   XS_Command := "HMI_CMD_SCH1".ES,
                   OS_Status => "STATUS_SCH1".ES);
   END_IF;
   #SF_BSN3_ES(IB1In := "Sfty_Status".BSN3_ES.Flt,   // "STD_DI_Mon"
               IB1Inv := "STDLog0",
               IB1Ack := "STATUS_Zone200".Mode.Specific.Ack,
               IB1AlmSupp := "STDLog0",
               XS_Parameter := "HMI_PARAM_BSN3".ES,
               XS_Command := "HMI_CMD_BSN3".ES,
               OS_Status => "STATUS_BSN3".ES,
               ENO => #_w3);
   IF #_w3 THEN
       #SF_BSN4_5_ES(IB1In := "Sfty_Status".BSN4_5_ES.Flt,   // "STD_DI_Mon"
                     IB1Inv := "STDLog0",
                     IB1Ack := "STATUS_Zone300".Mode.Specific.Ack,
                     IB1AlmSupp := "STDLog0",
                     XS_Parameter := "HMI_PARAM_BSN4".ES,
                     XS_Command := "HMI_CMD_BSN4".ES,
                     OS_Status => "STATUS_BSN4".ES);
   END_IF;
   #SF_THM1_ES(IB1In := "Sfty_Status".THM1_ES.Flt,   // "STD_DI_Mon"
               IB1Inv := "STDLog0",
               IB1Ack := "STATUS_Zone400".Mode.Specific.Ack,
               IB1AlmSupp := "STDLog0",
               XS_Parameter := "HMI_PARAM_THM1".ES,
               XS_Command := "HMI_CMD_THM1".ES,
               OS_Status => "STATUS_THM1".ES,
               ENO => #_w4);
   IF #_w4 THEN
       #SF_THM2_ES(IB1In := "Sfty_Status".THM2_ES.Flt,   // "STD_DI_Mon"
                   IB1Inv := "STDLog0",
                   IB1Ack := "STATUS_Zone400".Mode.Specific.Ack,
                   IB1AlmSupp := "STDLog0",
                   XS_Parameter := "HMI_PARAM_THM2".ES,
                   XS_Command := "HMI_CMD_THM2".ES,
                   OS_Status => "STATUS_THM2".ES);
   END_IF;
END_REGION

REGION Network 38: *************** Alarms estop buttons ***************
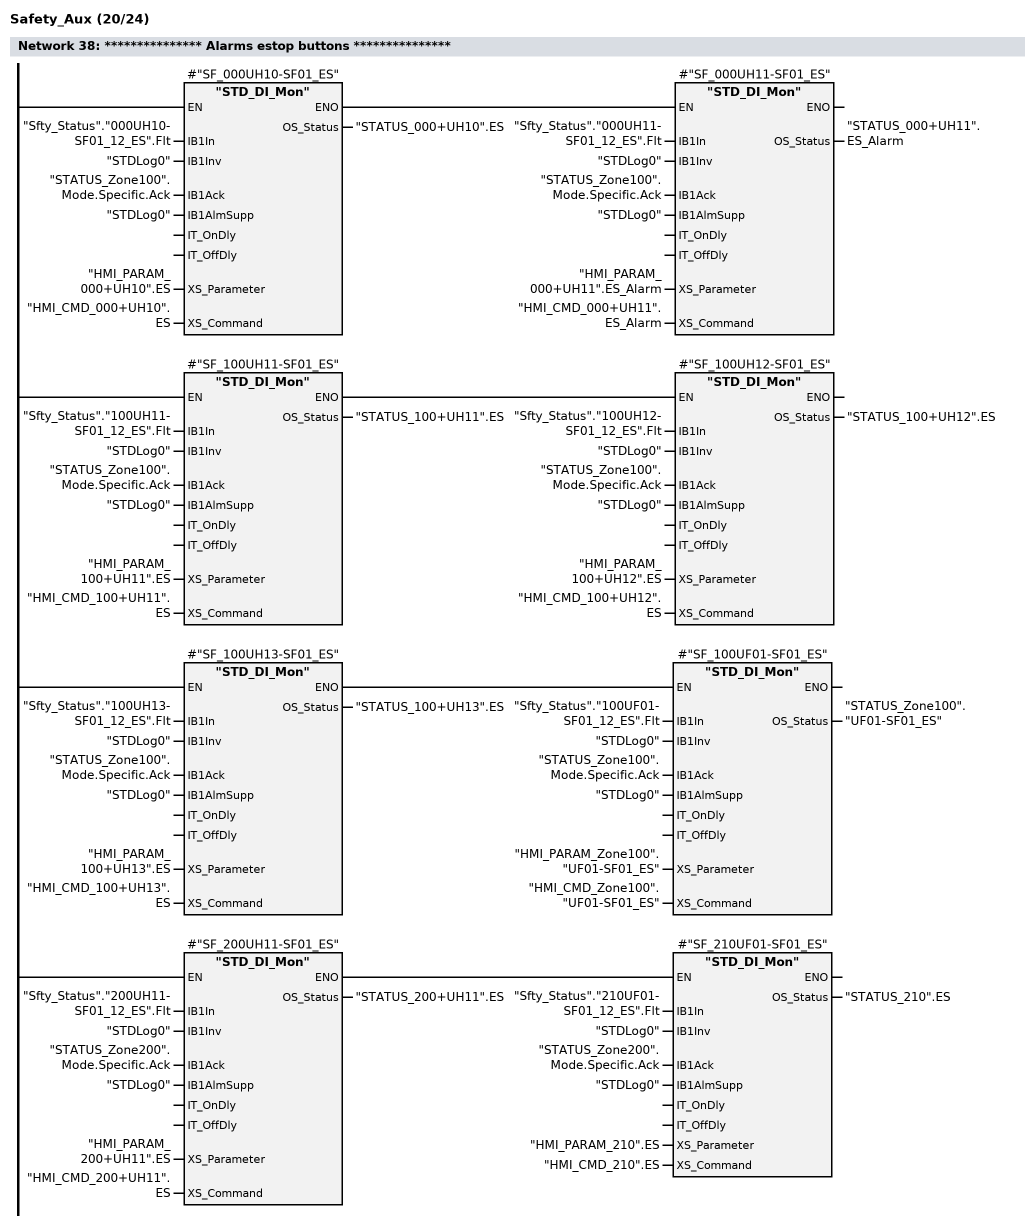
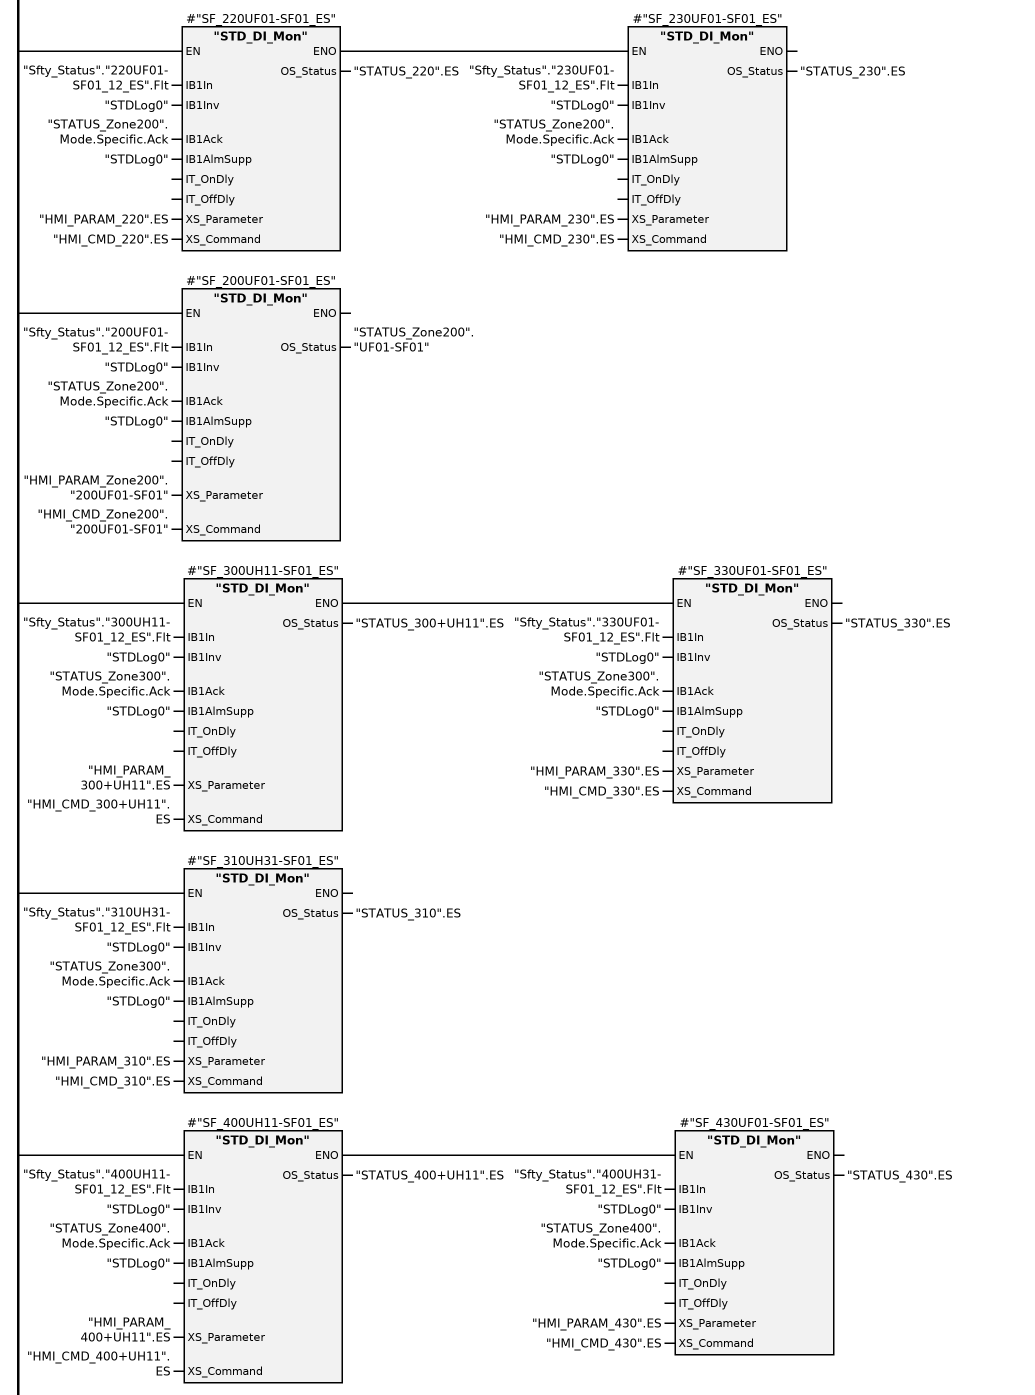
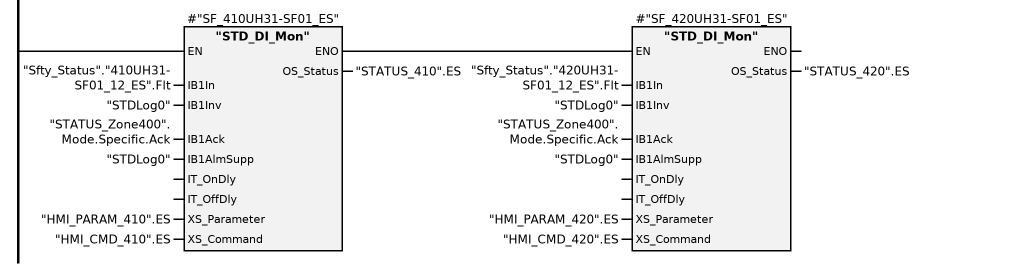
   RUNG wire#powerrail
      #"SF_000UH10-SF01_ES"(IB1In := "Sfty_Status"."000UH10-SF01_12_ES".Flt, IB1Inv := "STDLog0", IB1Ack := "STATUS_Zone100".Mode.Specific.Ack, IB1AlmSupp := "STDLog0", IT_OnDly :=, IT_OffDly :=, XS_Parameter := "HMI_PARAM_000+UH10".ES, XS_Command := "HMI_CMD_000+UH10".ES, OS_Status => "STATUS_000+UH10".ES)
      #"SF_000UH11-SF01_ES"(IB1In := "Sfty_Status"."000UH11-SF01_12_ES".Flt, IB1Inv := "STDLog0", IB1Ack := "STATUS_Zone100".Mode.Specific.Ack, IB1AlmSupp := "STDLog0", IT_OnDly :=, IT_OffDly :=, XS_Parameter := "HMI_PARAM_000+UH11".ES_Alarm, XS_Command := "HMI_CMD_000+UH11".ES_Alarm, OS_Status => "STATUS_000+UH11".ES_Alarm)
   END_RUNG
   RUNG wire#powerrail
      #"SF_100UH11-SF01_ES"(IB1In := "Sfty_Status"."100UH11-SF01_12_ES".Flt, IB1Inv := "STDLog0", IB1Ack := "STATUS_Zone100".Mode.Specific.Ack, IB1AlmSupp := "STDLog0", IT_OnDly :=, IT_OffDly :=, XS_Parameter := "HMI_PARAM_100+UH11".ES, XS_Command := "HMI_CMD_100+UH11".ES, OS_Status => "STATUS_100+UH11".ES)
      #"SF_100UH12-SF01_ES"(IB1In := "Sfty_Status"."100UH12-SF01_12_ES".Flt, IB1Inv := "STDLog0", IB1Ack := "STATUS_Zone100".Mode.Specific.Ack, IB1AlmSupp := "STDLog0", IT_OnDly :=, IT_OffDly :=, XS_Parameter := "HMI_PARAM_100+UH12".ES, XS_Command := "HMI_CMD_100+UH12".ES, OS_Status => "STATUS_100+UH12".ES)
   END_RUNG
   RUNG wire#powerrail
      #"SF_100UH13-SF01_ES"(IB1In := "Sfty_Status"."100UH13-SF01_12_ES".Flt, IB1Inv := "STDLog0", IB1Ack := "STATUS_Zone100".Mode.Specific.Ack, IB1AlmSupp := "STDLog0", IT_OnDly :=, IT_OffDly :=, XS_Parameter := "HMI_PARAM_100+UH13".ES, XS_Command := "HMI_CMD_100+UH13".ES, OS_Status => "STATUS_100+UH13".ES)
      #"SF_100UF01-SF01_ES"(IB1In := "Sfty_Status"."100UF01-SF01_12_ES".Flt, IB1Inv := "STDLog0", IB1Ack := "STATUS_Zone100".Mode.Specific.Ack, IB1AlmSupp := "STDLog0", IT_OnDly :=, IT_OffDly :=, XS_Parameter := "HMI_PARAM_Zone100"."UF01-SF01_ES", XS_Command := "HMI_CMD_Zone100"."UF01-SF01_ES", OS_Status => "STATUS_Zone100"."UF01-SF01_ES")
   END_RUNG
   RUNG wire#powerrail
      #"SF_200UH11-SF01_ES"(IB1In := "Sfty_Status"."200UH11-SF01_12_ES".Flt, IB1Inv := "STDLog0", IB1Ack := "STATUS_Zone200".Mode.Specific.Ack, IB1AlmSupp := "STDLog0", IT_OnDly :=, IT_OffDly :=, XS_Parameter := "HMI_PARAM_200+UH11".ES, XS_Command := "HMI_CMD_200+UH11".ES, OS_Status => "STATUS_200+UH11".ES)
      #"SF_210UF01-SF01_ES"(IB1In := "Sfty_Status"."210UF01-SF01_12_ES".Flt, IB1Inv := "STDLog0", IB1Ack := "STATUS_Zone200".Mode.Specific.Ack, IB1AlmSupp := "STDLog0", IT_OnDly :=, IT_OffDly :=, XS_Parameter := "HMI_PARAM_210".ES, XS_Command := "HMI_CMD_210".ES, OS_Status => "STATUS_210".ES)
   END_RUNG
   RUNG wire#powerrail
      #"SF_220UF01-SF01_ES"(IB1In := "Sfty_Status"."220UF01-SF01_12_ES".Flt, IB1Inv := "STDLog0", IB1Ack := "STATUS_Zone200".Mode.Specific.Ack, IB1AlmSupp := "STDLog0", IT_OnDly :=, IT_OffDly :=, XS_Parameter := "HMI_PARAM_220".ES, XS_Command := "HMI_CMD_220".ES, OS_Status => "STATUS_220".ES)
      #"SF_230UF01-SF01_ES"(IB1In := "Sfty_Status"."230UF01-SF01_12_ES".Flt, IB1Inv := "STDLog0", IB1Ack := "STATUS_Zone200".Mode.Specific.Ack, IB1AlmSupp := "STDLog0", IT_OnDly :=, IT_OffDly :=, XS_Parameter := "HMI_PARAM_230".ES, XS_Command := "HMI_CMD_230".ES, OS_Status => "STATUS_230".ES)
   END_RUNG
   RUNG wire#powerrail
      #"SF_200UF01-SF01_ES"(IB1In := "Sfty_Status"."200UF01-SF01_12_ES".Flt, IB1Inv := "STDLog0", IB1Ack := "STATUS_Zone200".Mode.Specific.Ack, IB1AlmSupp := "STDLog0", IT_OnDly :=, IT_OffDly :=, XS_Parameter := "HMI_PARAM_Zone200"."200UF01-SF01", XS_Command := "HMI_CMD_Zone200"."200UF01-SF01", OS_Status => "STATUS_Zone200"."UF01-SF01")
   END_RUNG
   RUNG wire#powerrail
      #"SF_300UH11-SF01_ES"(IB1In := "Sfty_Status"."300UH11-SF01_12_ES".Flt, IB1Inv := "STDLog0", IB1Ack := "STATUS_Zone300".Mode.Specific.Ack, IB1AlmSupp := "STDLog0", IT_OnDly :=, IT_OffDly :=, XS_Parameter := "HMI_PARAM_300+UH11".ES, XS_Command := "HMI_CMD_300+UH11".ES, OS_Status => "STATUS_300+UH11".ES)
      #"SF_330UF01-SF01_ES"(IB1In := "Sfty_Status"."330UF01-SF01_12_ES".Flt, IB1Inv := "STDLog0", IB1Ack := "STATUS_Zone300".Mode.Specific.Ack, IB1AlmSupp := "STDLog0", IT_OnDly :=, IT_OffDly :=, XS_Parameter := "HMI_PARAM_330".ES, XS_Command := "HMI_CMD_330".ES, OS_Status => "STATUS_330".ES)
   END_RUNG
   RUNG wire#powerrail
      #"SF_310UH31-SF01_ES"(IB1In := "Sfty_Status"."310UH31-SF01_12_ES".Flt, IB1Inv := "STDLog0", IB1Ack := "STATUS_Zone300".Mode.Specific.Ack, IB1AlmSupp := "STDLog0", IT_OnDly :=, IT_OffDly :=, XS_Parameter := "HMI_PARAM_310".ES, XS_Command := "HMI_CMD_310".ES, OS_Status => "STATUS_310".ES)
   END_RUNG
   RUNG wire#powerrail
      #"SF_400UH11-SF01_ES"(IB1In := "Sfty_Status"."400UH11-SF01_12_ES".Flt, IB1Inv := "STDLog0", IB1Ack := "STATUS_Zone400".Mode.Specific.Ack, IB1AlmSupp := "STDLog0", IT_OnDly :=, IT_OffDly :=, XS_Parameter := "HMI_PARAM_400+UH11".ES, XS_Command := "HMI_CMD_400+UH11".ES, OS_Status => "STATUS_400+UH11".ES)
      #"SF_430UF01-SF01_ES"(IB1In := "Sfty_Status"."400UH31-SF01_12_ES".Flt, IB1Inv := "STDLog0", IB1Ack := "STATUS_Zone400".Mode.Specific.Ack, IB1AlmSupp := "STDLog0", IT_OnDly :=, IT_OffDly :=, XS_Parameter := "HMI_PARAM_430".ES, XS_Command := "HMI_CMD_430".ES, OS_Status => "STATUS_430".ES)
   END_RUNG
   RUNG wire#powerrail
      #"SF_410UH31-SF01_ES"(IB1In := "Sfty_Status"."410UH31-SF01_12_ES".Flt, IB1Inv := "STDLog0", IB1Ack := "STATUS_Zone400".Mode.Specific.Ack, IB1AlmSupp := "STDLog0", IT_OnDly :=, IT_OffDly :=, XS_Parameter := "HMI_PARAM_410".ES, XS_Command := "HMI_CMD_410".ES, OS_Status => "STATUS_410".ES)
      #"SF_420UH31-SF01_ES"(IB1In := "Sfty_Status"."420UH31-SF01_12_ES".Flt, IB1Inv := "STDLog0", IB1Ack := "STATUS_Zone400".Mode.Specific.Ack, IB1AlmSupp := "STDLog0", IT_OnDly :=, IT_OffDly :=, XS_Parameter := "HMI_PARAM_420".ES, XS_Command := "HMI_CMD_420".ES, OS_Status => "STATUS_420".ES)
   END_RUNG
   // the same network as SCL:
   #"SF_000UH10-SF01_ES"(IB1In := "Sfty_Status"."000UH10-SF01_12_ES".Flt,   // "STD_DI_Mon"
                         IB1Inv := "STDLog0",
                         IB1Ack := "STATUS_Zone100".Mode.Specific.Ack,
                         IB1AlmSupp := "STDLog0",
                         XS_Parameter := "HMI_PARAM_000+UH10".ES,
                         XS_Command := "HMI_CMD_000+UH10".ES,
                         OS_Status => "STATUS_000+UH10".ES,
                         ENO => #_w1);
   IF #_w1 THEN
       #"SF_000UH11-SF01_ES"(IB1In := "Sfty_Status"."000UH11-SF01_12_ES".Flt,   // "STD_DI_Mon"
                             IB1Inv := "STDLog0",
                             IB1Ack := "STATUS_Zone100".Mode.Specific.Ack,
                             IB1AlmSupp := "STDLog0",
                             XS_Parameter := "HMI_PARAM_000+UH11".ES_Alarm,
                             XS_Command := "HMI_CMD_000+UH11".ES_Alarm,
                             OS_Status => "STATUS_000+UH11".ES_Alarm);
   END_IF;
   #"SF_100UH11-SF01_ES"(IB1In := "Sfty_Status"."100UH11-SF01_12_ES".Flt,   // "STD_DI_Mon"
                         IB1Inv := "STDLog0",
                         IB1Ack := "STATUS_Zone100".Mode.Specific.Ack,
                         IB1AlmSupp := "STDLog0",
                         XS_Parameter := "HMI_PARAM_100+UH11".ES,
                         XS_Command := "HMI_CMD_100+UH11".ES,
                         OS_Status => "STATUS_100+UH11".ES,
                         ENO => #_w2);
   IF #_w2 THEN
       #"SF_100UH12-SF01_ES"(IB1In := "Sfty_Status"."100UH12-SF01_12_ES".Flt,   // "STD_DI_Mon"
                             IB1Inv := "STDLog0",
                             IB1Ack := "STATUS_Zone100".Mode.Specific.Ack,
                             IB1AlmSupp := "STDLog0",
                             XS_Parameter := "HMI_PARAM_100+UH12".ES,
                             XS_Command := "HMI_CMD_100+UH12".ES,
                             OS_Status => "STATUS_100+UH12".ES);
   END_IF;
   #"SF_100UH13-SF01_ES"(IB1In := "Sfty_Status"."100UH13-SF01_12_ES".Flt,   // "STD_DI_Mon"
                         IB1Inv := "STDLog0",
                         IB1Ack := "STATUS_Zone100".Mode.Specific.Ack,
                         IB1AlmSupp := "STDLog0",
                         XS_Parameter := "HMI_PARAM_100+UH13".ES,
                         XS_Command := "HMI_CMD_100+UH13".ES,
                         OS_Status => "STATUS_100+UH13".ES,
                         ENO => #_w3);
   IF #_w3 THEN
       #"SF_100UF01-SF01_ES"(IB1In := "Sfty_Status"."100UF01-SF01_12_ES".Flt,   // "STD_DI_Mon"
                             IB1Inv := "STDLog0",
                             IB1Ack := "STATUS_Zone100".Mode.Specific.Ack,
                             IB1AlmSupp := "STDLog0",
                             XS_Parameter := "HMI_PARAM_Zone100"."UF01-SF01_ES",
                             XS_Command := "HMI_CMD_Zone100"."UF01-SF01_ES",
                             OS_Status => "STATUS_Zone100"."UF01-SF01_ES");
   END_IF;
   #"SF_200UH11-SF01_ES"(IB1In := "Sfty_Status"."200UH11-SF01_12_ES".Flt,   // "STD_DI_Mon"
                         IB1Inv := "STDLog0",
                         IB1Ack := "STATUS_Zone200".Mode.Specific.Ack,
                         IB1AlmSupp := "STDLog0",
                         XS_Parameter := "HMI_PARAM_200+UH11".ES,
                         XS_Command := "HMI_CMD_200+UH11".ES,
                         OS_Status => "STATUS_200+UH11".ES,
                         ENO => #_w4);
   IF #_w4 THEN
       #"SF_210UF01-SF01_ES"(IB1In := "Sfty_Status"."210UF01-SF01_12_ES".Flt,   // "STD_DI_Mon"
                             IB1Inv := "STDLog0",
                             IB1Ack := "STATUS_Zone200".Mode.Specific.Ack,
                             IB1AlmSupp := "STDLog0",
                             XS_Parameter := "HMI_PARAM_210".ES,
                             XS_Command := "HMI_CMD_210".ES,
                             OS_Status => "STATUS_210".ES);
   END_IF;
   #"SF_220UF01-SF01_ES"(IB1In := "Sfty_Status"."220UF01-SF01_12_ES".Flt,   // "STD_DI_Mon"
                         IB1Inv := "STDLog0",
                         IB1Ack := "STATUS_Zone200".Mode.Specific.Ack,
                         IB1AlmSupp := "STDLog0",
                         XS_Parameter := "HMI_PARAM_220".ES,
                         XS_Command := "HMI_CMD_220".ES,
                         OS_Status => "STATUS_220".ES,
                         ENO => #_w5);
   IF #_w5 THEN
       #"SF_230UF01-SF01_ES"(IB1In := "Sfty_Status"."230UF01-SF01_12_ES".Flt,   // "STD_DI_Mon"
                             IB1Inv := "STDLog0",
                             IB1Ack := "STATUS_Zone200".Mode.Specific.Ack,
                             IB1AlmSupp := "STDLog0",
                             XS_Parameter := "HMI_PARAM_230".ES,
                             XS_Command := "HMI_CMD_230".ES,
                             OS_Status => "STATUS_230".ES);
   END_IF;
   #"SF_200UF01-SF01_ES"(IB1In := "Sfty_Status"."200UF01-SF01_12_ES".Flt,   // "STD_DI_Mon"
                         IB1Inv := "STDLog0",
                         IB1Ack := "STATUS_Zone200".Mode.Specific.Ack,
                         IB1AlmSupp := "STDLog0",
                         XS_Parameter := "HMI_PARAM_Zone200"."200UF01-SF01",
                         XS_Command := "HMI_CMD_Zone200"."200UF01-SF01",
                         OS_Status => "STATUS_Zone200"."UF01-SF01");
   #"SF_300UH11-SF01_ES"(IB1In := "Sfty_Status"."300UH11-SF01_12_ES".Flt,   // "STD_DI_Mon"
                         IB1Inv := "STDLog0",
                         IB1Ack := "STATUS_Zone300".Mode.Specific.Ack,
                         IB1AlmSupp := "STDLog0",
                         XS_Parameter := "HMI_PARAM_300+UH11".ES,
                         XS_Command := "HMI_CMD_300+UH11".ES,
                         OS_Status => "STATUS_300+UH11".ES,
                         ENO => #_w6);
   IF #_w6 THEN
       #"SF_330UF01-SF01_ES"(IB1In := "Sfty_Status"."330UF01-SF01_12_ES".Flt,   // "STD_DI_Mon"
                             IB1Inv := "STDLog0",
                             IB1Ack := "STATUS_Zone300".Mode.Specific.Ack,
                             IB1AlmSupp := "STDLog0",
                             XS_Parameter := "HMI_PARAM_330".ES,
                             XS_Command := "HMI_CMD_330".ES,
                             OS_Status => "STATUS_330".ES);
   END_IF;
   #"SF_310UH31-SF01_ES"(IB1In := "Sfty_Status"."310UH31-SF01_12_ES".Flt,   // "STD_DI_Mon"
                         IB1Inv := "STDLog0",
                         IB1Ack := "STATUS_Zone300".Mode.Specific.Ack,
                         IB1AlmSupp := "STDLog0",
                         XS_Parameter := "HMI_PARAM_310".ES,
                         XS_Command := "HMI_CMD_310".ES,
                         OS_Status => "STATUS_310".ES);
   #"SF_400UH11-SF01_ES"(IB1In := "Sfty_Status"."400UH11-SF01_12_ES".Flt,   // "STD_DI_Mon"
                         IB1Inv := "STDLog0",
                         IB1Ack := "STATUS_Zone400".Mode.Specific.Ack,
                         IB1AlmSupp := "STDLog0",
                         XS_Parameter := "HMI_PARAM_400+UH11".ES,
                         XS_Command := "HMI_CMD_400+UH11".ES,
                         OS_Status => "STATUS_400+UH11".ES,
                         ENO => #_w7);
   IF #_w7 THEN
       #"SF_430UF01-SF01_ES"(IB1In := "Sfty_Status"."400UH31-SF01_12_ES".Flt,   // "STD_DI_Mon"
                             IB1Inv := "STDLog0",
                             IB1Ack := "STATUS_Zone400".Mode.Specific.Ack,
                             IB1AlmSupp := "STDLog0",
                             XS_Parameter := "HMI_PARAM_430".ES,
                             XS_Command := "HMI_CMD_430".ES,
                             OS_Status => "STATUS_430".ES);
   END_IF;
   #"SF_410UH31-SF01_ES"(IB1In := "Sfty_Status"."410UH31-SF01_12_ES".Flt,   // "STD_DI_Mon"
                         IB1Inv := "STDLog0",
                         IB1Ack := "STATUS_Zone400".Mode.Specific.Ack,
                         IB1AlmSupp := "STDLog0",
                         XS_Parameter := "HMI_PARAM_410".ES,
                         XS_Command := "HMI_CMD_410".ES,
                         OS_Status => "STATUS_410".ES,
                         ENO => #_w8);
   IF #_w8 THEN
       #"SF_420UH31-SF01_ES"(IB1In := "Sfty_Status"."420UH31-SF01_12_ES".Flt,   // "STD_DI_Mon"
                             IB1Inv := "STDLog0",
                             IB1Ack := "STATUS_Zone400".Mode.Specific.Ack,
                             IB1AlmSupp := "STDLog0",
                             XS_Parameter := "HMI_PARAM_420".ES,
                             XS_Command := "HMI_CMD_420".ES,
                             OS_Status => "STATUS_420".ES);
   END_IF;
END_REGION

REGION Network 39: *************** Alarms estop buttons gates ***************
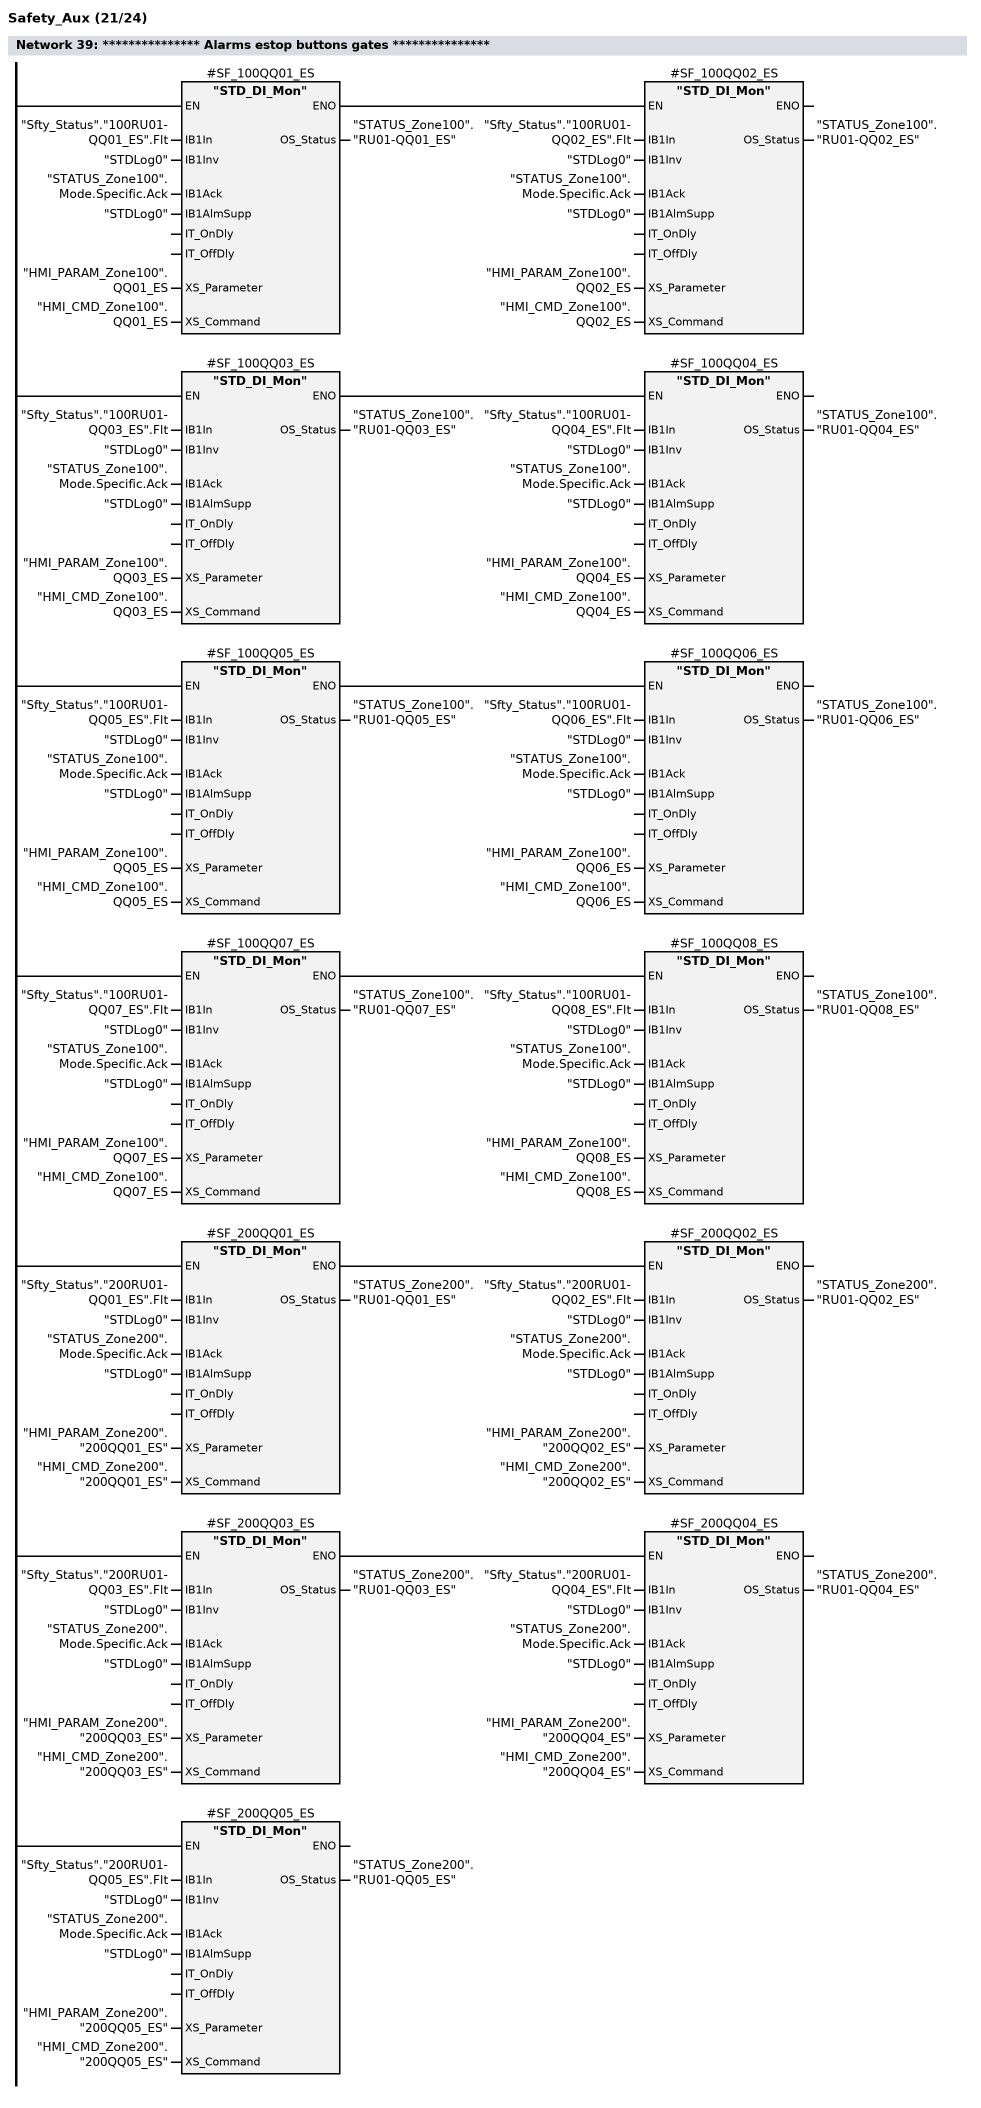
   RUNG wire#powerrail
      #SF_100QQ01_ES(IB1In := "Sfty_Status"."100RU01-QQ01_ES".Flt, IB1Inv := "STDLog0", IB1Ack := "STATUS_Zone100".Mode.Specific.Ack, IB1AlmSupp := "STDLog0", IT_OnDly :=, IT_OffDly :=, XS_Parameter := "HMI_PARAM_Zone100".QQ01_ES, XS_Command := "HMI_CMD_Zone100".QQ01_ES, OS_Status => "STATUS_Zone100"."RU01-QQ01_ES")
      #SF_100QQ02_ES(IB1In := "Sfty_Status"."100RU01-QQ02_ES".Flt, IB1Inv := "STDLog0", IB1Ack := "STATUS_Zone100".Mode.Specific.Ack, IB1AlmSupp := "STDLog0", IT_OnDly :=, IT_OffDly :=, XS_Parameter := "HMI_PARAM_Zone100".QQ02_ES, XS_Command := "HMI_CMD_Zone100".QQ02_ES, OS_Status => "STATUS_Zone100"."RU01-QQ02_ES")
   END_RUNG
   RUNG wire#powerrail
      #SF_100QQ03_ES(IB1In := "Sfty_Status"."100RU01-QQ03_ES".Flt, IB1Inv := "STDLog0", IB1Ack := "STATUS_Zone100".Mode.Specific.Ack, IB1AlmSupp := "STDLog0", IT_OnDly :=, IT_OffDly :=, XS_Parameter := "HMI_PARAM_Zone100".QQ03_ES, XS_Command := "HMI_CMD_Zone100".QQ03_ES, OS_Status => "STATUS_Zone100"."RU01-QQ03_ES")
      #SF_100QQ04_ES(IB1In := "Sfty_Status"."100RU01-QQ04_ES".Flt, IB1Inv := "STDLog0", IB1Ack := "STATUS_Zone100".Mode.Specific.Ack, IB1AlmSupp := "STDLog0", IT_OnDly :=, IT_OffDly :=, XS_Parameter := "HMI_PARAM_Zone100".QQ04_ES, XS_Command := "HMI_CMD_Zone100".QQ04_ES, OS_Status => "STATUS_Zone100"."RU01-QQ04_ES")
   END_RUNG
   RUNG wire#powerrail
      #SF_100QQ05_ES(IB1In := "Sfty_Status"."100RU01-QQ05_ES".Flt, IB1Inv := "STDLog0", IB1Ack := "STATUS_Zone100".Mode.Specific.Ack, IB1AlmSupp := "STDLog0", IT_OnDly :=, IT_OffDly :=, XS_Parameter := "HMI_PARAM_Zone100".QQ05_ES, XS_Command := "HMI_CMD_Zone100".QQ05_ES, OS_Status => "STATUS_Zone100"."RU01-QQ05_ES")
      #SF_100QQ06_ES(IB1In := "Sfty_Status"."100RU01-QQ06_ES".Flt, IB1Inv := "STDLog0", IB1Ack := "STATUS_Zone100".Mode.Specific.Ack, IB1AlmSupp := "STDLog0", IT_OnDly :=, IT_OffDly :=, XS_Parameter := "HMI_PARAM_Zone100".QQ06_ES, XS_Command := "HMI_CMD_Zone100".QQ06_ES, OS_Status => "STATUS_Zone100"."RU01-QQ06_ES")
   END_RUNG
   RUNG wire#powerrail
      #SF_100QQ07_ES(IB1In := "Sfty_Status"."100RU01-QQ07_ES".Flt, IB1Inv := "STDLog0", IB1Ack := "STATUS_Zone100".Mode.Specific.Ack, IB1AlmSupp := "STDLog0", IT_OnDly :=, IT_OffDly :=, XS_Parameter := "HMI_PARAM_Zone100".QQ07_ES, XS_Command := "HMI_CMD_Zone100".QQ07_ES, OS_Status => "STATUS_Zone100"."RU01-QQ07_ES")
      #SF_100QQ08_ES(IB1In := "Sfty_Status"."100RU01-QQ08_ES".Flt, IB1Inv := "STDLog0", IB1Ack := "STATUS_Zone100".Mode.Specific.Ack, IB1AlmSupp := "STDLog0", IT_OnDly :=, IT_OffDly :=, XS_Parameter := "HMI_PARAM_Zone100".QQ08_ES, XS_Command := "HMI_CMD_Zone100".QQ08_ES, OS_Status => "STATUS_Zone100"."RU01-QQ08_ES")
   END_RUNG
   RUNG wire#powerrail
      #SF_200QQ01_ES(IB1In := "Sfty_Status"."200RU01-QQ01_ES".Flt, IB1Inv := "STDLog0", IB1Ack := "STATUS_Zone200".Mode.Specific.Ack, IB1AlmSupp := "STDLog0", IT_OnDly :=, IT_OffDly :=, XS_Parameter := "HMI_PARAM_Zone200"."200QQ01_ES", XS_Command := "HMI_CMD_Zone200"."200QQ01_ES", OS_Status => "STATUS_Zone200"."RU01-QQ01_ES")
      #SF_200QQ02_ES(IB1In := "Sfty_Status"."200RU01-QQ02_ES".Flt, IB1Inv := "STDLog0", IB1Ack := "STATUS_Zone200".Mode.Specific.Ack, IB1AlmSupp := "STDLog0", IT_OnDly :=, IT_OffDly :=, XS_Parameter := "HMI_PARAM_Zone200"."200QQ02_ES", XS_Command := "HMI_CMD_Zone200"."200QQ02_ES", OS_Status => "STATUS_Zone200"."RU01-QQ02_ES")
   END_RUNG
   RUNG wire#powerrail
      #SF_200QQ03_ES(IB1In := "Sfty_Status"."200RU01-QQ03_ES".Flt, IB1Inv := "STDLog0", IB1Ack := "STATUS_Zone200".Mode.Specific.Ack, IB1AlmSupp := "STDLog0", IT_OnDly :=, IT_OffDly :=, XS_Parameter := "HMI_PARAM_Zone200"."200QQ03_ES", XS_Command := "HMI_CMD_Zone200"."200QQ03_ES", OS_Status => "STATUS_Zone200"."RU01-QQ03_ES")
      #SF_200QQ04_ES(IB1In := "Sfty_Status"."200RU01-QQ04_ES".Flt, IB1Inv := "STDLog0", IB1Ack := "STATUS_Zone200".Mode.Specific.Ack, IB1AlmSupp := "STDLog0", IT_OnDly :=, IT_OffDly :=, XS_Parameter := "HMI_PARAM_Zone200"."200QQ04_ES", XS_Command := "HMI_CMD_Zone200"."200QQ04_ES", OS_Status => "STATUS_Zone200"."RU01-QQ04_ES")
   END_RUNG
   RUNG wire#powerrail
      #SF_200QQ05_ES(IB1In := "Sfty_Status"."200RU01-QQ05_ES".Flt, IB1Inv := "STDLog0", IB1Ack := "STATUS_Zone200".Mode.Specific.Ack, IB1AlmSupp := "STDLog0", IT_OnDly :=, IT_OffDly :=, XS_Parameter := "HMI_PARAM_Zone200"."200QQ05_ES", XS_Command := "HMI_CMD_Zone200"."200QQ05_ES", OS_Status => "STATUS_Zone200"."RU01-QQ05_ES")
   END_RUNG
   // the same network as SCL:
   #SF_100QQ01_ES(IB1In := "Sfty_Status"."100RU01-QQ01_ES".Flt,   // "STD_DI_Mon"
                  IB1Inv := "STDLog0",
                  IB1Ack := "STATUS_Zone100".Mode.Specific.Ack,
                  IB1AlmSupp := "STDLog0",
                  XS_Parameter := "HMI_PARAM_Zone100".QQ01_ES,
                  XS_Command := "HMI_CMD_Zone100".QQ01_ES,
                  OS_Status => "STATUS_Zone100"."RU01-QQ01_ES",
                  ENO => #_w1);
   IF #_w1 THEN
       #SF_100QQ02_ES(IB1In := "Sfty_Status"."100RU01-QQ02_ES".Flt,   // "STD_DI_Mon"
                      IB1Inv := "STDLog0",
                      IB1Ack := "STATUS_Zone100".Mode.Specific.Ack,
                      IB1AlmSupp := "STDLog0",
                      XS_Parameter := "HMI_PARAM_Zone100".QQ02_ES,
                      XS_Command := "HMI_CMD_Zone100".QQ02_ES,
                      OS_Status => "STATUS_Zone100"."RU01-QQ02_ES");
   END_IF;
   #SF_100QQ03_ES(IB1In := "Sfty_Status"."100RU01-QQ03_ES".Flt,   // "STD_DI_Mon"
                  IB1Inv := "STDLog0",
                  IB1Ack := "STATUS_Zone100".Mode.Specific.Ack,
                  IB1AlmSupp := "STDLog0",
                  XS_Parameter := "HMI_PARAM_Zone100".QQ03_ES,
                  XS_Command := "HMI_CMD_Zone100".QQ03_ES,
                  OS_Status => "STATUS_Zone100"."RU01-QQ03_ES",
                  ENO => #_w2);
   IF #_w2 THEN
       #SF_100QQ04_ES(IB1In := "Sfty_Status"."100RU01-QQ04_ES".Flt,   // "STD_DI_Mon"
                      IB1Inv := "STDLog0",
                      IB1Ack := "STATUS_Zone100".Mode.Specific.Ack,
                      IB1AlmSupp := "STDLog0",
                      XS_Parameter := "HMI_PARAM_Zone100".QQ04_ES,
                      XS_Command := "HMI_CMD_Zone100".QQ04_ES,
                      OS_Status => "STATUS_Zone100"."RU01-QQ04_ES");
   END_IF;
   #SF_100QQ05_ES(IB1In := "Sfty_Status"."100RU01-QQ05_ES".Flt,   // "STD_DI_Mon"
                  IB1Inv := "STDLog0",
                  IB1Ack := "STATUS_Zone100".Mode.Specific.Ack,
                  IB1AlmSupp := "STDLog0",
                  XS_Parameter := "HMI_PARAM_Zone100".QQ05_ES,
                  XS_Command := "HMI_CMD_Zone100".QQ05_ES,
                  OS_Status => "STATUS_Zone100"."RU01-QQ05_ES",
                  ENO => #_w3);
   IF #_w3 THEN
       #SF_100QQ06_ES(IB1In := "Sfty_Status"."100RU01-QQ06_ES".Flt,   // "STD_DI_Mon"
                      IB1Inv := "STDLog0",
                      IB1Ack := "STATUS_Zone100".Mode.Specific.Ack,
                      IB1AlmSupp := "STDLog0",
                      XS_Parameter := "HMI_PARAM_Zone100".QQ06_ES,
                      XS_Command := "HMI_CMD_Zone100".QQ06_ES,
                      OS_Status => "STATUS_Zone100"."RU01-QQ06_ES");
   END_IF;
   #SF_100QQ07_ES(IB1In := "Sfty_Status"."100RU01-QQ07_ES".Flt,   // "STD_DI_Mon"
                  IB1Inv := "STDLog0",
                  IB1Ack := "STATUS_Zone100".Mode.Specific.Ack,
                  IB1AlmSupp := "STDLog0",
                  XS_Parameter := "HMI_PARAM_Zone100".QQ07_ES,
                  XS_Command := "HMI_CMD_Zone100".QQ07_ES,
                  OS_Status => "STATUS_Zone100"."RU01-QQ07_ES",
                  ENO => #_w4);
   IF #_w4 THEN
       #SF_100QQ08_ES(IB1In := "Sfty_Status"."100RU01-QQ08_ES".Flt,   // "STD_DI_Mon"
                      IB1Inv := "STDLog0",
                      IB1Ack := "STATUS_Zone100".Mode.Specific.Ack,
                      IB1AlmSupp := "STDLog0",
                      XS_Parameter := "HMI_PARAM_Zone100".QQ08_ES,
                      XS_Command := "HMI_CMD_Zone100".QQ08_ES,
                      OS_Status => "STATUS_Zone100"."RU01-QQ08_ES");
   END_IF;
   #SF_200QQ01_ES(IB1In := "Sfty_Status"."200RU01-QQ01_ES".Flt,   // "STD_DI_Mon"
                  IB1Inv := "STDLog0",
                  IB1Ack := "STATUS_Zone200".Mode.Specific.Ack,
                  IB1AlmSupp := "STDLog0",
                  XS_Parameter := "HMI_PARAM_Zone200"."200QQ01_ES",
                  XS_Command := "HMI_CMD_Zone200"."200QQ01_ES",
                  OS_Status => "STATUS_Zone200"."RU01-QQ01_ES",
                  ENO => #_w5);
   IF #_w5 THEN
       #SF_200QQ02_ES(IB1In := "Sfty_Status"."200RU01-QQ02_ES".Flt,   // "STD_DI_Mon"
                      IB1Inv := "STDLog0",
                      IB1Ack := "STATUS_Zone200".Mode.Specific.Ack,
                      IB1AlmSupp := "STDLog0",
                      XS_Parameter := "HMI_PARAM_Zone200"."200QQ02_ES",
                      XS_Command := "HMI_CMD_Zone200"."200QQ02_ES",
                      OS_Status => "STATUS_Zone200"."RU01-QQ02_ES");
   END_IF;
   #SF_200QQ03_ES(IB1In := "Sfty_Status"."200RU01-QQ03_ES".Flt,   // "STD_DI_Mon"
                  IB1Inv := "STDLog0",
                  IB1Ack := "STATUS_Zone200".Mode.Specific.Ack,
                  IB1AlmSupp := "STDLog0",
                  XS_Parameter := "HMI_PARAM_Zone200"."200QQ03_ES",
                  XS_Command := "HMI_CMD_Zone200"."200QQ03_ES",
                  OS_Status => "STATUS_Zone200"."RU01-QQ03_ES",
                  ENO => #_w6);
   IF #_w6 THEN
       #SF_200QQ04_ES(IB1In := "Sfty_Status"."200RU01-QQ04_ES".Flt,   // "STD_DI_Mon"
                      IB1Inv := "STDLog0",
                      IB1Ack := "STATUS_Zone200".Mode.Specific.Ack,
                      IB1AlmSupp := "STDLog0",
                      XS_Parameter := "HMI_PARAM_Zone200"."200QQ04_ES",
                      XS_Command := "HMI_CMD_Zone200"."200QQ04_ES",
                      OS_Status => "STATUS_Zone200"."RU01-QQ04_ES");
   END_IF;
   #SF_200QQ05_ES(IB1In := "Sfty_Status"."200RU01-QQ05_ES".Flt,   // "STD_DI_Mon"
                  IB1Inv := "STDLog0",
                  IB1Ack := "STATUS_Zone200".Mode.Specific.Ack,
                  IB1AlmSupp := "STDLog0",
                  XS_Parameter := "HMI_PARAM_Zone200"."200QQ05_ES",
                  XS_Command := "HMI_CMD_Zone200"."200QQ05_ES",
                  OS_Status => "STATUS_Zone200"."RU01-QQ05_ES");
END_REGION

